LIN {X 0,Y 523.895,Z 313.853,A -85,B 0,C 180,E1 -4885.421,E2 -4885.421} C_VEL
LIN {X 0,Y 523.902,Z 313.843,A -85,B 0,C 180,E1 -4888.002,E2 -4888.002} C_VEL
LIN {X 0,Y 523.925,Z 313.85,A -85,B 0,C 180,E1 -4890.853,E2 -4890.853} C_VEL
LIN {X 0,Y 523.919,Z 313.846,A -85,B 0,C 180,E1 -4893.73,E2 -4893.73} C_VEL
LIN {X 0,Y 523.893,Z 313.85,A -85,B 0,C 180,E1 -4896.402,E2 -4896.402} C_VEL
LIN {X 0,Y 523.91,Z 313.85,A -85,B 0,C 180,E1 -4899.085,E2 -4899.085} C_VEL
LIN {X 0,Y 523.942,Z 313.841,A -85,B 0,C 180,E1 -4902.119,E2 -4902.119} C_VEL
LIN {X 0,Y 523.933,Z 313.845,A -85,B 0,C 180,E1 -4905.311,E2 -4905.311} C_VEL
LIN {X 0,Y 523.907,Z 313.852,A -85,B 0,C 180,E1 -4906.866,E2 -4906.866} C_VEL
LIN {X 0,Y 523.227,Z 313.935,A -85,B 0,C 180,E1 -4907.294,E2 -4907.294} C_VEL
LIN {X 0,Y 520.387,Z 314.288,A -85,B 0,C 180,E1 -4907.962,E2 -4907.962} C_VEL
LIN {X 0,Y 517.542,Z 314.646,A -85,B 0,C 180,E1 -4908.638,E2 -4908.638} C_VEL
LIN {X 0,Y 516.872,Z 314.727,A -85,B 0,C 180,E1 -4909.074,E2 -4909.074} C_VEL
LIN {X 0,Y 516.91,Z 314.812,A -85,B 0,C 180,E1 -4909.879,E2 -4909.879} C_VEL
LIN {X 0,Y 518.209,Z 321.592,A -85,B 0,C 180,E1 -4911.166,E2 -4911.166} C_VEL
LIN {X 0,Y 518.031,Z 330.95,A -85,B 0,C 180,E1 -4912.826,E2 -4912.826} C_VEL
LIN {X 0,Y 518.003,Z 334.606,A -85,B 0,C 180,E1 -4913.443,E2 -4913.443} C_VEL
LIN {X 0,Y 520.419,Z 345.939,A -85,B 0,C 180,E1 -4913.696,E2 -4913.696} C_VEL
LIN {X 0,Y 519.712,Z 470.939,A -85,B 0,C 180,E1 -4915.474,E2 -4915.474} C_VEL
LIN {X 0,Y 519.472,Z 485.199,A -85,B 0,C 180,E1 -4915.836,E2 -4915.836} C_VEL
LIN {X 0,Y 519.165,Z 498.963,A -85,B 0,C 180,E1 -4916.347,E2 -4916.347} C_VEL
LIN {X 0,Y 518.789,Z 511.827,A -85,B 0,C 180,E1 -4916.982,E2 -4916.982} C_VEL
LIN {X 0,Y 518.377,Z 523.912,A -85,B 0,C 180,E1 -4917.736,E2 -4917.736} C_VEL
LIN {X 0,Y 517.97,Z 535.685,A -85,B 0,C 180,E1 -4918.645,E2 -4918.645} C_VEL
LIN {X 0,Y 517.554,Z 547.16,A -85,B 0,C 180,E1 -4919.727,E2 -4919.727} C_VEL
LIN {X 0,Y 517.208,Z 557.645,A -85,B 0,C 180,E1 -4920.937,E2 -4920.937} C_VEL
LIN {X 0,Y 516.873,Z 567.085,A -85,B 0,C 180,E1 -4922.278,E2 -4922.278} C_VEL
LIN {X 0,Y 516.634,Z 574.914,A -85,B 0,C 180,E1 -4923.646,E2 -4923.646} C_VEL
LIN {X 0,Y 516.429,Z 581.367,A -85,B 0,C 180,E1 -4925.048,E2 -4925.048} C_VEL
LIN {X 0,Y 516.394,Z 586.053,A -85,B 0,C 180,E1 -4926.33,E2 -4926.33} C_VEL
LIN {X 0,Y 516.291,Z 590.061,A -85,B 0,C 180,E1 -4927.765,E2 -4927.765} C_VEL
LIN {X 0,Y 516.188,Z 592.955,A -85,B 0,C 180,E1 -4929.269,E2 -4929.269} C_VEL
LIN {X 0,Y 516.2,Z 594.008,A -85,B 0,C 180,E1 -4930.101,E2 -4930.101} C_VEL
LIN {X 0,Y 516.169,Z 594.998,A -85,B 0,C 180,E1 -4931.751,E2 -4931.751} C_VEL
LIN {X 0,Y 516.164,Z 594.545,A -85,B 0,C 180,E1 -4933.386,E2 -4933.386} C_VEL
LIN {X 0,Y 516.216,Z 592.673,A -85,B 0,C 180,E1 -4935.009,E2 -4935.009} C_VEL
LIN {X 0,Y 516.273,Z 589.339,A -85,B 0,C 180,E1 -4936.62,E2 -4936.62} C_VEL
LIN {X 0,Y 516.396,Z 584.476,A -85,B 0,C 180,E1 -4938.221,E2 -4938.221} C_VEL
LIN {X 0,Y 516.474,Z 579.801,A -85,B 0,C 180,E1 -4939.415,E2 -4939.415} C_VEL
LIN {X 0,Y 516.689,Z 572.998,A -85,B 0,C 180,E1 -4940.804,E2 -4940.804} C_VEL
LIN {X 0,Y 516.94,Z 564.592,A -85,B 0,C 180,E1 -4942.187,E2 -4942.187} C_VEL
LIN {X 0,Y 517.273,Z 555.841,A -85,B 0,C 180,E1 -4943.369,E2 -4943.369} C_VEL
LIN {X 0,Y 517.611,Z 545.305,A -85,B 0,C 180,E1 -4944.547,E2 -4944.547} C_VEL
LIN {X 0,Y 517.958,Z 534.696,A -85,B 0,C 180,E1 -4945.526,E2 -4945.526} C_VEL
LIN {X 0,Y 518.401,Z 523.103,A -85,B 0,C 180,E1 -4946.406,E2 -4946.406} C_VEL
LIN {X 0,Y 518.815,Z 510.389,A -85,B 0,C 180,E1 -4947.186,E2 -4947.186} C_VEL
LIN {X 0,Y 519.208,Z 497.174,A -85,B 0,C 180,E1 -4947.819,E2 -4947.819} C_VEL
LIN {X 0,Y 519.498,Z 483.55,A -85,B 0,C 180,E1 -4948.305,E2 -4948.305} C_VEL
LIN {X 0,Y 519.723,Z 469.332,A -85,B 0,C 180,E1 -4948.645,E2 -4948.645} C_VEL
LIN {X 0,Y 520.457,Z 346.248,A -85,B 0,C 180,E1 -4950.386,E2 -4950.386} C_VEL
LIN {X 0,Y 517.964,Z 334.247,A -85,B 0,C 180,E1 -4950.669,E2 -4950.669} C_VEL
LIN {X 0,Y 518.252,Z 321.48,A -85,B 0,C 180,E1 -4952.916,E2 -4952.916} C_VEL
LIN {X 0,Y 516.918,Z 314.722,A -85,B 0,C 180,E1 -4954.216,E2 -4954.216} C_VEL
LIN {X 0,Y 516.981,Z 314.712,A -85,B 0,C 180,E1 -4956.244,E2 -4956.244} C_VEL
LIN {X 0,Y 516.932,Z 314.723,A -85,B 0,C 180,E1 -4959.39,E2 -4959.39} C_VEL
LIN {X 0,Y 516.95,Z 314.714,A -85,B 0,C 180,E1 -4961.807,E2 -4961.807} C_VEL
LIN {X 0,Y 516.934,Z 314.721,A -85,B 0,C 180,E1 -4965.143,E2 -4965.143} C_VEL
LIN {X 0,Y 516.91,Z 314.716,A -85,B 0,C 180,E1 -4968.223,E2 -4968.223} C_VEL
LIN {X 0,Y 516.902,Z 314.72,A -85,B 0,C 180,E1 -4970.702,E2 -4970.702} C_VEL
LIN {X 0,Y 516.882,Z 314.72,A -85,B 0,C 180,E1 -4974.074,E2 -4974.074} C_VEL
LIN {X 0,Y 516.835,Z 314.729,A -85,B 0,C 180,E1 -4976.663,E2 -4976.663} C_VEL
LIN {X 0,Y 516.878,Z 314.722,A -85,B 0,C 180,E1 -4979.518,E2 -4979.518} C_VEL
LIN {X 0,Y 516.862,Z 314.725,A -85,B 0,C 180,E1 -4982.538,E2 -4982.538} C_VEL
LIN {X 0,Y 516.847,Z 314.727,A -85,B 0,C 180,E1 -4985.327,E2 -4985.327} C_VEL
LIN {X 0,Y 516.859,Z 314.73,A -85,B 0,C 180,E1 -4988.718,E2 -4988.718} C_VEL
LIN {X 0,Y 516.841,Z 314.725,A -85,B 0,C 180,E1 -4991.783,E2 -4991.783} C_VEL
LIN {X 0,Y 516.895,Z 314.723,A -85,B 0,C 180,E1 -4995.007,E2 -4995.007} C_VEL
LIN {X 0,Y 516.845,Z 314.729,A -85,B 0,C 180,E1 -4998.408,E2 -4998.408} C_VEL
LIN {X 0,Y 516.854,Z 314.724,A -85,B 0,C 180,E1 -5001.282,E2 -5001.282} C_VEL
LIN {X 0,Y 516.849,Z 314.732,A -85,B 0,C 180,E1 -5004.674,E2 -5004.674} C_VEL
LIN {X 0,Y 516.892,Z 314.719,A -85,B 0,C 180,E1 -5007.458,E2 -5007.458} C_VEL
LIN {X 0,Y 516.889,Z 314.725,A -85,B 0,C 180,E1 -5010.694,E2 -5010.694} C_VEL
LIN {X 0,Y 516.879,Z 314.721,A -85,B 0,C 180,E1 -5013.819,E2 -5013.819} C_VEL
LIN {X 0,Y 516.842,Z 314.728,A -85,B 0,C 180,E1 -5016.775,E2 -5016.775} C_VEL
LIN {X 0,Y 516.928,Z 314.716,A -85,B 0,C 180,E1 -5019.736,E2 -5019.736} C_VEL
LIN {X 0,Y 516.866,Z 314.726,A -85,B 0,C 180,E1 -5022.594,E2 -5022.594} C_VEL
LIN {X 0,Y 516.934,Z 314.714,A -85,B 0,C 180,E1 -5025.03,E2 -5025.03} C_VEL
LIN {X 0,Y 516.969,Z 314.718,A -85,B 0,C 180,E1 -5028.234,E2 -5028.234} C_VEL
LIN {X 0,Y 516.955,Z 314.711,A -85,B 0,C 180,E1 -5031.4,E2 -5031.4} C_VEL
LIN {X 0,Y 517.02,Z 314.705,A -85,B 0,C 180,E1 -5034.54,E2 -5034.54} C_VEL
LIN {X 0,Y 517.082,Z 314.699,A -85,B 0,C 180,E1 -5037.663,E2 -5037.663} C_VEL
LIN {X 0,Y 517.093,Z 314.694,A -85,B 0,C 180,E1 -5040.779,E2 -5040.779} C_VEL
LIN {X 0,Y 516.976,Z 314.708,A -85,B 0,C 180,E1 -5043.117,E2 -5043.117} C_VEL
LIN {X 0,Y 516.991,Z 314.71,A -85,B 0,C 180,E1 -5046.244,E2 -5046.244} C_VEL
LIN {X 0,Y 516.967,Z 314.71,A -85,B 0,C 180,E1 -5048.601,E2 -5048.601} C_VEL
LIN {X 0,Y 516.955,Z 314.72,A -85,B 0,C 180,E1 -5051.807,E2 -5051.807} C_VEL
LIN {X 0,Y 516.948,Z 314.713,A -85,B 0,C 180,E1 -5055.146,E2 -5055.146} C_VEL
LIN {X 0,Y 516.928,Z 314.716,A -85,B 0,C 180,E1 -5058.222,E2 -5058.222} C_VEL
LIN {X 0,Y 516.916,Z 314.715,A -85,B 0,C 180,E1 -5060.702,E2 -5060.702} C_VEL
LIN {X 0,Y 516.894,Z 314.721,A -85,B 0,C 180,E1 -5064.073,E2 -5064.073} C_VEL
LIN {X 0,Y 516.926,Z 314.714,A -85,B 0,C 180,E1 -5066.658,E2 -5066.658} C_VEL
LIN {X 0,Y 516.914,Z 314.725,A -85,B 0,C 180,E1 -5069.524,E2 -5069.524} C_VEL
LIN {X 0,Y 516.899,Z 314.718,A -85,B 0,C 180,E1 -5072.543,E2 -5072.543} C_VEL
LIN {X 0,Y 516.868,Z 314.73,A -85,B 0,C 180,E1 -5075.329,E2 -5075.329} C_VEL
LIN {X 0,Y 516.882,Z 314.721,A -85,B 0,C 180,E1 -5077.943,E2 -5077.943} C_VEL
LIN {X 0,Y 516.887,Z 314.721,A -85,B 0,C 180,E1 -5080.742,E2 -5080.742} C_VEL
LIN {X 0,Y 516.887,Z 314.722,A -85,B 0,C 180,E1 -5082.831,E2 -5082.831} C_VEL
LIN {X 0,Y 516.927,Z 314.72,A -85,B 0,C 180,E1 -5085.01,E2 -5085.01} C_VEL
LIN {X 0,Y 516.917,Z 314.716,A -85,B 0,C 180,E1 -5088.399,E2 -5088.399} C_VEL
LIN {X 0,Y 516.886,Z 314.726,A -85,B 0,C 180,E1 -5091.284,E2 -5091.284} C_VEL
LIN {X 0,Y 516.876,Z 314.721,A -85,B 0,C 180,E1 -5094.219,E2 -5094.219} C_VEL
LIN {X 0,Y 516.899,Z 314.727,A -85,B 0,C 180,E1 -5097.053,E2 -5097.053} C_VEL
LIN {X 0,Y 516.891,Z 314.724,A -85,B 0,C 180,E1 -5099.796,E2 -5099.796} C_VEL
LIN {X 0,Y 516.926,Z 314.725,A -85,B 0,C 180,E1 -5102.905,E2 -5102.905} C_VEL
LIN {X 0,Y 516.96,Z 314.746,A -85,B 0,C 180,E1 -5103.344,E2 -5103.344} C_VEL
LIN {X 0,Y 519.314,Z 326.551,A -85,B 0,C 180,E1 -5105.195,E2 -5105.195} C_VEL
LIN {X 0,Y 518.6,Z 348.488,A -85,B 0,C 180,E1 -5108.328,E2 -5108.328} C_VEL
LIN {X 0,Y 518.011,Z 369.079,A -85,B 0,C 180,E1 -5111.222,E2 -5111.222} C_VEL
LIN {X 0,Y 518.022,Z 370.448,A -85,B 0,C 180,E1 -5111.379,E2 -5111.379} C_VEL
LIN {X 0,Y 520.349,Z 384.488,A -85,B 0,C 180,E1 -5111.665,E2 -5111.665} C_VEL
LIN {X 0,Y 519.632,Z 508.513,A -85,B 0,C 180,E1 -5113.423,E2 -5113.423} C_VEL
LIN {X 0,Y 519.349,Z 523,A -85,B 0,C 180,E1 -5113.788,E2 -5113.788} C_VEL
LIN {X 0,Y 519.043,Z 536.545,A -85,B 0,C 180,E1 -5114.287,E2 -5114.287} C_VEL
LIN {X 0,Y 518.616,Z 550.559,A -85,B 0,C 180,E1 -5114.979,E2 -5114.979} C_VEL
LIN {X 0,Y 518.19,Z 563.097,A -85,B 0,C 180,E1 -5115.769,E2 -5115.769} C_VEL
LIN {X 0,Y 517.789,Z 574.555,A -85,B 0,C 180,E1 -5116.659,E2 -5116.659} C_VEL
LIN {X 0,Y 517.429,Z 585.048,A -85,B 0,C 180,E1 -5117.643,E2 -5117.643} C_VEL
LIN {X 0,Y 517.129,Z 595.568,A -85,B 0,C 180,E1 -5118.833,E2 -5118.833} C_VEL
LIN {X 0,Y 516.807,Z 604.214,A -85,B 0,C 180,E1 -5120.015,E2 -5120.015} C_VEL
LIN {X 0,Y 516.591,Z 612.5,A -85,B 0,C 180,E1 -5121.393,E2 -5121.393} C_VEL
LIN {X 0,Y 516.447,Z 618.297,A -85,B 0,C 180,E1 -5122.571,E2 -5122.571} C_VEL
LIN {X 0,Y 516.365,Z 623.051,A -85,B 0,C 180,E1 -5123.748,E2 -5123.748} C_VEL
LIN {X 0,Y 516.306,Z 626.901,A -85,B 0,C 180,E1 -5124.923,E2 -5124.923} C_VEL
LIN {X 0,Y 516.325,Z 629.869,A -85,B 0,C 180,E1 -5126.097,E2 -5126.097} C_VEL
LIN {X 0,Y 516.259,Z 632.583,A -85,B 0,C 180,E1 -5127.659,E2 -5127.659} C_VEL
LIN {X 0,Y 516.157,Z 633.926,A -85,B 0,C 180,E1 -5129.219,E2 -5129.219} C_VEL
LIN {X 0,Y 516.157,Z 633.926,A -85,B 0,C 180,E1 -5130.779,E2 -5130.779} C_VEL
LIN {X 0,Y 516.259,Z 632.584,A -85,B 0,C 180,E1 -5132.34,E2 -5132.34} C_VEL
LIN {X 0,Y 516.324,Z 629.869,A -85,B 0,C 180,E1 -5133.902,E2 -5133.902} C_VEL
LIN {X 0,Y 516.366,Z 625.705,A -85,B 0,C 180,E1 -5135.466,E2 -5135.466} C_VEL
LIN {X 0,Y 516.401,Z 619.967,A -85,B 0,C 180,E1 -5137.035,E2 -5137.035} C_VEL
LIN {X 0,Y 516.582,Z 613.504,A -85,B 0,C 180,E1 -5138.409,E2 -5138.409} C_VEL
LIN {X 0,Y 516.76,Z 605.473,A -85,B 0,C 180,E1 -5139.787,E2 -5139.787} C_VEL
LIN {X 0,Y 517.069,Z 597.078,A -85,B 0,C 180,E1 -5140.969,E2 -5140.969} C_VEL
LIN {X 0,Y 517.388,Z 586.704,A -85,B 0,C 180,E1 -5142.183,E2 -5142.183} C_VEL
LIN {X 0,Y 517.738,Z 575.7,A -85,B 0,C 180,E1 -5143.241,E2 -5143.241} C_VEL
LIN {X 0,Y 518.14,Z 564.494,A -85,B 0,C 180,E1 -5144.131,E2 -5144.131} C_VEL
LIN {X 0,Y 518.543,Z 552.292,A -85,B 0,C 180,E1 -5144.922,E2 -5144.922} C_VEL
LIN {X 0,Y 518.966,Z 538.756,A -85,B 0,C 180,E1 -5145.613,E2 -5145.613} C_VEL
LIN {X 0,Y 519.283,Z 524.557,A -85,B 0,C 180,E1 -5146.159,E2 -5146.159} C_VEL
LIN {X 0,Y 519.563,Z 510.759,A -85,B 0,C 180,E1 -5146.527,E2 -5146.527} C_VEL
LIN {X 0,Y 519.766,Z 488.556,A -85,B 0,C 180,E1 -5146.874,E2 -5146.874} C_VEL
LIN {X 0,Y 520.331,Z 383.603,A -85,B 0,C 180,E1 -5148.347,E2 -5148.347} C_VEL
LIN {X 0,Y 517.954,Z 369.999,A -85,B 0,C 180,E1 -5148.634,E2 -5148.634} C_VEL
LIN {X 0,Y 518.61,Z 348.337,A -85,B 0,C 180,E1 -5151.67,E2 -5151.67} C_VEL
LIN {X 0,Y 519.25,Z 327.875,A -85,B 0,C 180,E1 -5154.594,E2 -5154.594} C_VEL
LIN {X 0,Y 518.84,Z 323.477,A -85,B 0,C 180,E1 -5155.256,E2 -5155.256} C_VEL
LIN {X 0,Y 516.957,Z 314.718,A -85,B 0,C 180,E1 -5156.655,E2 -5156.655} C_VEL
LIN {X 0,Y 516.909,Z 314.722,A -85,B 0,C 180,E1 -5159.523,E2 -5159.523} C_VEL
LIN {X 0,Y 516.895,Z 314.723,A -85,B 0,C 180,E1 -5162.543,E2 -5162.543} C_VEL
LIN {X 0,Y 516.88,Z 314.723,A -85,B 0,C 180,E1 -5165.331,E2 -5165.331} C_VEL
LIN {X 0,Y 516.878,Z 314.722,A -85,B 0,C 180,E1 -5167.942,E2 -5167.942} C_VEL
LIN {X 0,Y 516.9,Z 314.726,A -85,B 0,C 180,E1 -5170.739,E2 -5170.739} C_VEL
LIN {X 0,Y 516.878,Z 314.723,A -85,B 0,C 180,E1 -5173.902,E2 -5173.902} C_VEL
LIN {X 0,Y 516.878,Z 314.719,A -85,B 0,C 180,E1 -5176.106,E2 -5176.106} C_VEL
LIN {X 0,Y 516.912,Z 314.723,A -85,B 0,C 180,E1 -5178.397,E2 -5178.397} C_VEL
LIN {X 0,Y 516.877,Z 314.72,A -85,B 0,C 180,E1 -5181.284,E2 -5181.284} C_VEL
LIN {X 0,Y 516.883,Z 314.726,A -85,B 0,C 180,E1 -5184.22,E2 -5184.22} C_VEL
LIN {X 0,Y 516.89,Z 314.719,A -85,B 0,C 180,E1 -5187.052,E2 -5187.052} C_VEL
LIN {X 0,Y 516.895,Z 314.72,A -85,B 0,C 180,E1 -5189.796,E2 -5189.796} C_VEL
LIN {X 0,Y 516.924,Z 314.72,A -85,B 0,C 180,E1 -5192.467,E2 -5192.467} C_VEL
LIN {X 0,Y 516.897,Z 314.719,A -85,B 0,C 180,E1 -5195.071,E2 -5195.071} C_VEL
LIN {X 0,Y 516.878,Z 314.726,A -85,B 0,C 180,E1 -5198.462,E2 -5198.462} C_VEL
LIN {X 0,Y 516.894,Z 314.716,A -85,B 0,C 180,E1 -5200.954,E2 -5200.954} C_VEL
LIN {X 0,Y 516.904,Z 314.719,A -85,B 0,C 180,E1 -5203.41,E2 -5203.41} C_VEL
LIN {X 0,Y 516.885,Z 314.723,A -85,B 0,C 180,E1 -5205.833,E2 -5205.833} C_VEL
LIN {X 0,Y 516.957,Z 314.713,A -85,B 0,C 180,E1 -5208.233,E2 -5208.233} C_VEL
LIN {X 0,Y 516.954,Z 314.714,A -85,B 0,C 180,E1 -5211.399,E2 -5211.399} C_VEL
LIN {X 0,Y 516.989,Z 314.711,A -85,B 0,C 180,E1 -5213.756,E2 -5213.756} C_VEL
LIN {X 0,Y 516.962,Z 314.708,A -85,B 0,C 180,E1 -5216.883,E2 -5216.883} C_VEL
LIN {X 0,Y 517.08,Z 314.698,A -85,B 0,C 180,E1 -5219.221,E2 -5219.221} C_VEL
LIN {X 0,Y 517.063,Z 314.699,A -85,B 0,C 180,E1 -5222.337,E2 -5222.337} C_VEL
LIN {X 0,Y 516.97,Z 314.714,A -85,B 0,C 180,E1 -5225.46,E2 -5225.46} C_VEL
LIN {X 0,Y 516.914,Z 314.715,A -85,B 0,C 180,E1 -5228.601,E2 -5228.601} C_VEL
LIN {X 0,Y 516.942,Z 314.715,A -85,B 0,C 180,E1 -5231.807,E2 -5231.807} C_VEL
LIN {X 0,Y 516.924,Z 314.721,A -85,B 0,C 180,E1 -5235.142,E2 -5235.142} C_VEL
LIN {X 0,Y 516.865,Z 314.723,A -85,B 0,C 180,E1 -5238.224,E2 -5238.224} C_VEL
LIN {X 0,Y 516.89,Z 314.721,A -85,B 0,C 180,E1 -5240.702,E2 -5240.702} C_VEL
LIN {X 0,Y 516.845,Z 314.733,A -85,B 0,C 180,E1 -5243.224,E2 -5243.224} C_VEL
LIN {X 0,Y 516.888,Z 314.721,A -85,B 0,C 180,E1 -5246.186,E2 -5246.186} C_VEL
LIN {X 0,Y 516.893,Z 314.724,A -85,B 0,C 180,E1 -5249.306,E2 -5249.306} C_VEL
LIN {X 0,Y 516.884,Z 314.724,A -85,B 0,C 180,E1 -5252.543,E2 -5252.543} C_VEL
LIN {X 0,Y 516.855,Z 314.729,A -85,B 0,C 180,E1 -5255.33,E2 -5255.33} C_VEL
LIN {X 0,Y 516.87,Z 314.724,A -85,B 0,C 180,E1 -5257.943,E2 -5257.943} C_VEL
LIN {X 0,Y 516.874,Z 314.728,A -85,B 0,C 180,E1 -5260.742,E2 -5260.742} C_VEL
LIN {X 0,Y 516.873,Z 314.73,A -85,B 0,C 180,E1 -5262.832,E2 -5262.832} C_VEL
LIN {X 0,Y 516.886,Z 314.726,A -85,B 0,C 180,E1 -5265.007,E2 -5265.007} C_VEL
LIN {X 0,Y 516.905,Z 314.725,A -85,B 0,C 180,E1 -5268.399,E2 -5268.399} C_VEL
LIN {X 0,Y 516.872,Z 314.727,A -85,B 0,C 180,E1 -5269.074,E2 -5269.074} C_VEL
LIN {X 0,Y 516.621,Z 315.183,A -85,B 0,C 180,E1 -5269.504,E2 -5269.504} C_VEL
LIN {X 0,Y 515.985,Z 316.355,A -85,B 0,C 180,E1 -5269.915,E2 -5269.915} C_VEL
LIN {X 0,Y 514.111,Z 320.017,A -85,B 0,C 180,E1 -5270.678,E2 -5270.678} C_VEL
LIN {X 0,Y 511.532,Z 326.847,A -85,B 0,C 180,E1 -5271.783,E2 -5271.783} C_VEL
LIN {X 0,Y 511.257,Z 329.026,A -85,B 0,C 180,E1 -5272.164,E2 -5272.164} C_VEL
LIN {X 0,Y 511.074,Z 334.779,A -85,B 0,C 180,E1 -5273.179,E2 -5273.179} C_VEL
LIN {X 0,Y 513.686,Z 346.942,A -85,B 0,C 180,E1 -5273.458,E2 -5273.458} C_VEL
LIN {X 0,Y 512.919,Z 471.171,A -85,B 0,C 180,E1 -5275.249,E2 -5275.249} C_VEL
LIN {X 0,Y 512.66,Z 485.216,A -85,B 0,C 180,E1 -5275.608,E2 -5275.608} C_VEL
LIN {X 0,Y 512.349,Z 499.236,A -85,B 0,C 180,E1 -5276.135,E2 -5276.135} C_VEL
LIN {X 0,Y 511.895,Z 513.153,A -85,B 0,C 180,E1 -5276.836,E2 -5276.836} C_VEL
LIN {X 0,Y 511.478,Z 524.978,A -85,B 0,C 180,E1 -5277.597,E2 -5277.597} C_VEL
LIN {X 0,Y 511.033,Z 536.424,A -85,B 0,C 180,E1 -5278.501,E2 -5278.501} C_VEL
LIN {X 0,Y 510.588,Z 547.892,A -85,B 0,C 180,E1 -5279.606,E2 -5279.606} C_VEL
LIN {X 0,Y 510.249,Z 557.474,A -85,B 0,C 180,E1 -5280.729,E2 -5280.729} C_VEL
LIN {X 0,Y 509.903,Z 566.821,A -85,B 0,C 180,E1 -5282.056,E2 -5282.056} C_VEL
LIN {X 0,Y 509.617,Z 574.325,A -85,B 0,C 180,E1 -5283.358,E2 -5283.358} C_VEL
LIN {X 0,Y 509.427,Z 580.551,A -85,B 0,C 180,E1 -5284.681,E2 -5284.681} C_VEL
LIN {X 0,Y 509.321,Z 585.551,A -85,B 0,C 180,E1 -5286.006,E2 -5286.006} C_VEL
LIN {X 0,Y 509.189,Z 590.165,A -85,B 0,C 180,E1 -5287.63,E2 -5287.63} C_VEL
LIN {X 0,Y 509.119,Z 592.842,A -85,B 0,C 180,E1 -5288.968,E2 -5288.968} C_VEL
LIN {X 0,Y 509.121,Z 594.033,A -85,B 0,C 180,E1 -5289.831,E2 -5289.831} C_VEL
LIN {X 0,Y 509.085,Z 595.215,A -85,B 0,C 180,E1 -5291.488,E2 -5291.488} C_VEL
LIN {X 0,Y 509.128,Z 595.268,A -85,B 0,C 180,E1 -5292.322,E2 -5292.322} C_VEL
LIN {X 0,Y 509.046,Z 594.314,A -85,B 0,C 180,E1 -5293.972,E2 -5293.972} C_VEL
LIN {X 0,Y 509.161,Z 591.933,A -85,B 0,C 180,E1 -5295.615,E2 -5295.615} C_VEL
LIN {X 0,Y 509.238,Z 588.114,A -85,B 0,C 180,E1 -5297.244,E2 -5297.244} C_VEL
LIN {X 0,Y 509.344,Z 584.322,A -85,B 0,C 180,E1 -5298.424,E2 -5298.424} C_VEL
LIN {X 0,Y 509.455,Z 579.375,A -85,B 0,C 180,E1 -5299.67,E2 -5299.67} C_VEL
LIN {X 0,Y 509.635,Z 572.43,A -85,B 0,C 180,E1 -5301.076,E2 -5301.076} C_VEL
LIN {X 0,Y 509.973,Z 563.568,A -85,B 0,C 180,E1 -5302.518,E2 -5302.518} C_VEL
LIN {X 0,Y 510.304,Z 554.893,A -85,B 0,C 180,E1 -5303.675,E2 -5303.675} C_VEL
LIN {X 0,Y 510.717,Z 544.106,A -85,B 0,C 180,E1 -5304.869,E2 -5304.869} C_VEL
LIN {X 0,Y 511.111,Z 533.199,A -85,B 0,C 180,E1 -5305.861,E2 -5305.861} C_VEL
LIN {X 0,Y 511.596,Z 521.209,A -85,B 0,C 180,E1 -5306.752,E2 -5306.752} C_VEL
LIN {X 0,Y 512.078,Z 507.819,A -85,B 0,C 180,E1 -5307.543,E2 -5307.543} C_VEL
LIN {X 0,Y 512.445,Z 494.913,A -85,B 0,C 180,E1 -5308.134,E2 -5308.134} C_VEL
LIN {X 0,Y 512.725,Z 481.071,A -85,B 0,C 180,E1 -5308.602,E2 -5308.602} C_VEL
LIN {X 0,Y 512.975,Z 466.261,A -85,B 0,C 180,E1 -5308.925,E2 -5308.925} C_VEL
LIN {X 0,Y 513.668,Z 347.031,A -85,B 0,C 180,E1 -5310.63,E2 -5310.63} C_VEL
LIN {X 0,Y 511.048,Z 334.459,A -85,B 0,C 180,E1 -5310.936,E2 -5310.936} C_VEL
LIN {X 0,Y 511.341,Z 323.112,A -85,B 0,C 180,E1 -5312.955,E2 -5312.955} C_VEL
LIN {X 0,Y 509.902,Z 315.596,A -85,B 0,C 180,E1 -5314.398,E2 -5314.398} C_VEL
LIN {X 0,Y 509.973,Z 315.587,A -85,B 0,C 180,E1 -5317.145,E2 -5317.145} C_VEL
LIN {X 0,Y 509.843,Z 315.6,A -85,B 0,C 180,E1 -5320.324,E2 -5320.324} C_VEL
LIN {X 0,Y 509.867,Z 315.596,A -85,B 0,C 180,E1 -5322.742,E2 -5322.742} C_VEL
LIN {X 0,Y 509.843,Z 315.597,A -85,B 0,C 180,E1 -5326.004,E2 -5326.004} C_VEL
LIN {X 0,Y 509.855,Z 315.596,A -85,B 0,C 180,E1 -5328.485,E2 -5328.485} C_VEL
LIN {X 0,Y 509.843,Z 315.603,A -85,B 0,C 180,E1 -5331.003,E2 -5331.003} C_VEL
LIN {X 0,Y 509.816,Z 315.603,A -85,B 0,C 180,E1 -5333.565,E2 -5333.565} C_VEL
LIN {X 0,Y 509.812,Z 315.601,A -85,B 0,C 180,E1 -5336.357,E2 -5336.357} C_VEL
LIN {X 0,Y 509.829,Z 315.605,A -85,B 0,C 180,E1 -5338.848,E2 -5338.848} C_VEL
LIN {X 0,Y 509.786,Z 315.605,A -85,B 0,C 180,E1 -5341.593,E2 -5341.593} C_VEL
LIN {X 0,Y 509.826,Z 315.601,A -85,B 0,C 180,E1 -5344.416,E2 -5344.416} C_VEL
LIN {X 0,Y 509.773,Z 315.608,A -85,B 0,C 180,E1 -5347.345,E2 -5347.345} C_VEL
LIN {X 0,Y 509.811,Z 315.604,A -85,B 0,C 180,E1 -5350.385,E2 -5350.385} C_VEL
LIN {X 0,Y 509.789,Z 315.604,A -85,B 0,C 180,E1 -5353.576,E2 -5353.576} C_VEL
LIN {X 0,Y 509.789,Z 315.608,A -85,B 0,C 180,E1 -5356.425,E2 -5356.425} C_VEL
LIN {X 0,Y 509.791,Z 315.603,A -85,B 0,C 180,E1 -5359.614,E2 -5359.614} C_VEL
LIN {X 0,Y 509.772,Z 315.614,A -85,B 0,C 180,E1 -5362.656,E2 -5362.656} C_VEL
LIN {X 0,Y 509.838,Z 315.598,A -85,B 0,C 180,E1 -5365.801,E2 -5365.801} C_VEL
LIN {X 0,Y 509.837,Z 315.603,A -85,B 0,C 180,E1 -5368.722,E2 -5368.722} C_VEL
LIN {X 0,Y 509.823,Z 315.6,A -85,B 0,C 180,E1 -5371.153,E2 -5371.153} C_VEL
LIN {X 0,Y 509.848,Z 315.597,A -85,B 0,C 180,E1 -5373.826,E2 -5373.826} C_VEL
LIN {X 0,Y 509.809,Z 315.609,A -85,B 0,C 180,E1 -5376.436,E2 -5376.436} C_VEL
LIN {X 0,Y 509.906,Z 315.591,A -85,B 0,C 180,E1 -5379.845,E2 -5379.845} C_VEL
LIN {X 0,Y 509.848,Z 315.604,A -85,B 0,C 180,E1 -5382.347,E2 -5382.347} C_VEL
LIN {X 0,Y 509.885,Z 315.593,A -85,B 0,C 180,E1 -5384.818,E2 -5384.818} C_VEL
LIN {X 0,Y 509.903,Z 315.597,A -85,B 0,C 180,E1 -5388.125,E2 -5388.125} C_VEL
LIN {X 0,Y 509.903,Z 315.589,A -85,B 0,C 180,E1 -5391.28,E2 -5391.28} C_VEL
LIN {X 0,Y 509.971,Z 315.584,A -85,B 0,C 180,E1 -5394.464,E2 -5394.464} C_VEL
LIN {X 0,Y 510.052,Z 315.574,A -85,B 0,C 180,E1 -5397.631,E2 -5397.631} C_VEL
LIN {X 0,Y 510.063,Z 315.57,A -85,B 0,C 180,E1 -5400.79,E2 -5400.79} C_VEL
LIN {X 0,Y 509.92,Z 315.587,A -85,B 0,C 180,E1 -5403.161,E2 -5403.161} C_VEL
LIN {X 0,Y 509.939,Z 315.588,A -85,B 0,C 180,E1 -5406.33,E2 -5406.33} C_VEL
LIN {X 0,Y 509.913,Z 315.588,A -85,B 0,C 180,E1 -5408.72,E2 -5408.72} C_VEL
LIN {X 0,Y 509.908,Z 315.595,A -85,B 0,C 180,E1 -5411.932,E2 -5411.932} C_VEL
LIN {X 0,Y 509.898,Z 315.592,A -85,B 0,C 180,E1 -5415.242,E2 -5415.242} C_VEL
LIN {X 0,Y 509.885,Z 315.596,A -85,B 0,C 180,E1 -5417.998,E2 -5417.998} C_VEL
LIN {X 0,Y 509.854,Z 315.596,A -85,B 0,C 180,E1 -5421.002,E2 -5421.002} C_VEL
LIN {X 0,Y 509.826,Z 315.607,A -85,B 0,C 180,E1 -5423.564,E2 -5423.564} C_VEL
LIN {X 0,Y 509.914,Z 315.588,A -85,B 0,C 180,E1 -5426.378,E2 -5426.378} C_VEL
LIN {X 0,Y 509.878,Z 315.593,A -85,B 0,C 180,E1 -5428.844,E2 -5428.844} C_VEL
LIN {X 0,Y 509.824,Z 315.606,A -85,B 0,C 180,E1 -5431.59,E2 -5431.59} C_VEL
LIN {X 0,Y 509.85,Z 315.596,A -85,B 0,C 180,E1 -5434.414,E2 -5434.414} C_VEL
LIN {X 0,Y 509.811,Z 315.609,A -85,B 0,C 180,E1 -5437.342,E2 -5437.342} C_VEL
LIN {X 0,Y 509.842,Z 315.597,A -85,B 0,C 180,E1 -5440.382,E2 -5440.382} C_VEL
LIN {X 0,Y 509.828,Z 315.604,A -85,B 0,C 180,E1 -5443.062,E2 -5443.062} C_VEL
LIN {X 0,Y 509.834,Z 315.599,A -85,B 0,C 180,E1 -5445.792,E2 -5445.792} C_VEL
LIN {X 0,Y 509.859,Z 315.596,A -85,B 0,C 180,E1 -5448.574,E2 -5448.574} C_VEL
LIN {X 0,Y 509.855,Z 315.596,A -85,B 0,C 180,E1 -5451.786,E2 -5451.786} C_VEL
LIN {X 0,Y 509.835,Z 315.6,A -85,B 0,C 180,E1 -5454.622,E2 -5454.622} C_VEL
LIN {X 0,Y 509.865,Z 315.6,A -85,B 0,C 180,E1 -5457.481,E2 -5457.481} C_VEL
LIN {X 0,Y 509.862,Z 315.6,A -85,B 0,C 180,E1 -5460.274,E2 -5460.274} C_VEL
LIN {X 0,Y 509.911,Z 315.608,A -85,B 0,C 180,E1 -5463.116,E2 -5463.116} C_VEL
LIN {X 0,Y 512.392,Z 327.624,A -85,B 0,C 180,E1 -5465.034,E2 -5465.034} C_VEL
LIN {X 0,Y 511.764,Z 346.778,A -85,B 0,C 180,E1 -5467.811,E2 -5467.811} C_VEL
LIN {X 0,Y 511.165,Z 367.213,A -85,B 0,C 180,E1 -5470.732,E2 -5470.732} C_VEL
LIN {X 0,Y 511.049,Z 370.036,A -85,B 0,C 180,E1 -5471.114,E2 -5471.114} C_VEL
LIN {X 0,Y 513.603,Z 385.193,A -85,B 0,C 180,E1 -5471.429,E2 -5471.429} C_VEL
LIN {X 0,Y 512.803,Z 508.183,A -85,B 0,C 180,E1 -5473.196,E2 -5473.196} C_VEL
LIN {X 0,Y 512.514,Z 522.519,A -85,B 0,C 180,E1 -5473.56,E2 -5473.56} C_VEL
LIN {X 0,Y 512.181,Z 536.248,A -85,B 0,C 180,E1 -5474.071,E2 -5474.071} C_VEL
LIN {X 0,Y 511.732,Z 550.27,A -85,B 0,C 180,E1 -5474.772,E2 -5474.772} C_VEL
LIN {X 0,Y 511.266,Z 562.812,A -85,B 0,C 180,E1 -5475.572,E2 -5475.572} C_VEL
LIN {X 0,Y 510.808,Z 574.273,A -85,B 0,C 180,E1 -5476.473,E2 -5476.473} C_VEL
LIN {X 0,Y 510.446,Z 584.995,A -85,B 0,C 180,E1 -5477.494,E2 -5477.494} C_VEL
LIN {X 0,Y 510.1,Z 595.291,A -85,B 0,C 180,E1 -5478.677,E2 -5478.677} C_VEL
LIN {X 0,Y 509.745,Z 603.94,A -85,B 0,C 180,E1 -5479.875,E2 -5479.875} C_VEL
LIN {X 0,Y 509.536,Z 612.229,A -85,B 0,C 180,E1 -5481.273,E2 -5481.273} C_VEL
LIN {X 0,Y 509.37,Z 618.026,A -85,B 0,C 180,E1 -5482.468,E2 -5482.468} C_VEL
LIN {X 0,Y 509.262,Z 622.781,A -85,B 0,C 180,E1 -5483.661,E2 -5483.661} C_VEL
LIN {X 0,Y 509.236,Z 626.634,A -85,B 0,C 180,E1 -5484.853,E2 -5484.853} C_VEL
LIN {X 0,Y 509.218,Z 629.601,A -85,B 0,C 180,E1 -5486.042,E2 -5486.042} C_VEL
LIN {X 0,Y 509.188,Z 632.317,A -85,B 0,C 180,E1 -5487.626,E2 -5487.626} C_VEL
LIN {X 0,Y 509.071,Z 633.658,A -85,B 0,C 180,E1 -5489.208,E2 -5489.208} C_VEL
LIN {X 0,Y 509.071,Z 633.657,A -85,B 0,C 180,E1 -5490.79,E2 -5490.79} C_VEL
LIN {X 0,Y 509.187,Z 632.314,A -85,B 0,C 180,E1 -5492.372,E2 -5492.372} C_VEL
LIN {X 0,Y 509.218,Z 629.596,A -85,B 0,C 180,E1 -5493.956,E2 -5493.956} C_VEL
LIN {X 0,Y 509.282,Z 625.43,A -85,B 0,C 180,E1 -5495.543,E2 -5495.543} C_VEL
LIN {X 0,Y 509.326,Z 619.689,A -85,B 0,C 180,E1 -5497.133,E2 -5497.133} C_VEL
LIN {X 0,Y 509.504,Z 613.222,A -85,B 0,C 180,E1 -5498.527,E2 -5498.527} C_VEL
LIN {X 0,Y 509.723,Z 605.188,A -85,B 0,C 180,E1 -5499.924,E2 -5499.924} C_VEL
LIN {X 0,Y 510.028,Z 596.789,A -85,B 0,C 180,E1 -5501.122,E2 -5501.122} C_VEL
LIN {X 0,Y 510.402,Z 586.037,A -85,B 0,C 180,E1 -5502.393,E2 -5502.393} C_VEL
LIN {X 0,Y 510.781,Z 575.403,A -85,B 0,C 180,E1 -5503.425,E2 -5503.425} C_VEL
LIN {X 0,Y 511.224,Z 564.192,A -85,B 0,C 180,E1 -5504.326,E2 -5504.326} C_VEL
LIN {X 0,Y 511.646,Z 551.983,A -85,B 0,C 180,E1 -5505.128,E2 -5505.128} C_VEL
LIN {X 0,Y 512.119,Z 538.44,A -85,B 0,C 180,E1 -5505.827,E2 -5505.827} C_VEL
LIN {X 0,Y 512.458,Z 524.378,A -85,B 0,C 180,E1 -5506.375,E2 -5506.375} C_VEL
LIN {X 0,Y 512.742,Z 510.405,A -85,B 0,C 180,E1 -5506.753,E2 -5506.753} C_VEL
LIN {X 0,Y 512.957,Z 488.163,A -85,B 0,C 180,E1 -5507.105,E2 -5507.105} C_VEL
LIN {X 0,Y 513.613,Z 385.046,A -85,B 0,C 180,E1 -5508.57,E2 -5508.57} C_VEL
LIN {X 0,Y 511.047,Z 369.712,A -85,B 0,C 180,E1 -5508.896,E2 -5508.896} C_VEL
LIN {X 0,Y 511.705,Z 348.088,A -85,B 0,C 180,E1 -5511.978,E2 -5511.978} C_VEL
LIN {X 0,Y 512.383,Z 329.208,A -85,B 0,C 180,E1 -5514.715,E2 -5514.715} C_VEL
LIN {X 0,Y 511.866,Z 324.723,A -85,B 0,C 180,E1 -5515.407,E2 -5515.407} C_VEL
LIN {X 0,Y 509.903,Z 315.598,A -85,B 0,C 180,E1 -5516.925,E2 -5516.925} C_VEL
LIN {X 0,Y 509.855,Z 315.599,A -85,B 0,C 180,E1 -5519.75,E2 -5519.75} C_VEL
LIN {X 0,Y 509.872,Z 315.601,A -85,B 0,C 180,E1 -5522.773,E2 -5522.773} C_VEL
LIN {X 0,Y 509.84,Z 315.598,A -85,B 0,C 180,E1 -5525.58,E2 -5525.58} C_VEL
LIN {X 0,Y 509.848,Z 315.6,A -85,B 0,C 180,E1 -5528.337,E2 -5528.337} C_VEL
LIN {X 0,Y 509.861,Z 315.594,A -85,B 0,C 180,E1 -5531.424,E2 -5531.424} C_VEL
LIN {X 0,Y 509.852,Z 315.602,A -85,B 0,C 180,E1 -5534.667,E2 -5534.667} C_VEL
LIN {X 0,Y 509.856,Z 315.599,A -85,B 0,C 180,E1 -5538.102,E2 -5538.102} C_VEL
LIN {X 0,Y 509.842,Z 315.598,A -85,B 0,C 180,E1 -5540.647,E2 -5540.647} C_VEL
LIN {X 0,Y 509.829,Z 315.599,A -85,B 0,C 180,E1 -5543.647,E2 -5543.647} C_VEL
LIN {X 0,Y 509.855,Z 315.601,A -85,B 0,C 180,E1 -5546.539,E2 -5546.539} C_VEL
LIN {X 0,Y 509.844,Z 315.597,A -85,B 0,C 180,E1 -5549.334,E2 -5549.334} C_VEL
LIN {X 0,Y 509.889,Z 315.596,A -85,B 0,C 180,E1 -5552.054,E2 -5552.054} C_VEL
LIN {X 0,Y 509.867,Z 315.597,A -85,B 0,C 180,E1 -5554.703,E2 -5554.703} C_VEL
LIN {X 0,Y 509.818,Z 315.598,A -85,B 0,C 180,E1 -5557.457,E2 -5557.457} C_VEL
LIN {X 0,Y 509.909,Z 315.594,A -85,B 0,C 180,E1 -5559.844,E2 -5559.844} C_VEL
LIN {X 0,Y 509.875,Z 315.594,A -85,B 0,C 180,E1 -5563.174,E2 -5563.174} C_VEL
LIN {X 0,Y 509.854,Z 315.596,A -85,B 0,C 180,E1 -5565.634,E2 -5565.634} C_VEL
LIN {X 0,Y 509.903,Z 315.586,A -85,B 0,C 180,E1 -5568.874,E2 -5568.874} C_VEL
LIN {X 0,Y 509.941,Z 315.588,A -85,B 0,C 180,E1 -5572.078,E2 -5572.078} C_VEL
LIN {X 0,Y 509.965,Z 315.584,A -85,B 0,C 180,E1 -5574.464,E2 -5574.464} C_VEL
LIN {X 0,Y 510.036,Z 315.577,A -85,B 0,C 180,E1 -5577.631,E2 -5577.631} C_VEL
LIN {X 0,Y 510.022,Z 315.578,A -85,B 0,C 180,E1 -5580,E2 -5580} C_VEL
LIN {X 0,Y 510.034,Z 315.574,A -85,B 0,C 180,E1 -5582.369,E2 -5582.369} C_VEL
LIN {X 0,Y 509.922,Z 315.592,A -85,B 0,C 180,E1 -5585.536,E2 -5585.536} C_VEL
LIN {X 0,Y 509.866,Z 315.597,A -85,B 0,C 180,E1 -5587.923,E2 -5587.923} C_VEL
LIN {X 0,Y 509.896,Z 315.595,A -85,B 0,C 180,E1 -5591.126,E2 -5591.126} C_VEL
LIN {X 0,Y 509.828,Z 315.6,A -85,B 0,C 180,E1 -5594.367,E2 -5594.367} C_VEL
LIN {X 0,Y 509.808,Z 315.602,A -85,B 0,C 180,E1 -5596.828,E2 -5596.828} C_VEL
LIN {X 0,Y 509.896,Z 315.591,A -85,B 0,C 180,E1 -5600.156,E2 -5600.156} C_VEL
LIN {X 0,Y 509.807,Z 315.606,A -85,B 0,C 180,E1 -5603.564,E2 -5603.564} C_VEL
LIN {X 0,Y 509.865,Z 315.596,A -85,B 0,C 180,E1 -5606.37,E2 -5606.37} C_VEL
LIN {X 0,Y 509.841,Z 315.6,A -85,B 0,C 180,E1 -5609.752,E2 -5609.752} C_VEL
LIN {X 0,Y 509.857,Z 315.6,A -85,B 0,C 180,E1 -5612.773,E2 -5612.773} C_VEL
LIN {X 0,Y 509.815,Z 315.603,A -85,B 0,C 180,E1 -5615.579,E2 -5615.579} C_VEL
LIN {X 0,Y 509.84,Z 315.601,A -85,B 0,C 180,E1 -5618.338,E2 -5618.338} C_VEL
LIN {X 0,Y 509.846,Z 315.598,A -85,B 0,C 180,E1 -5621.426,E2 -5621.426} C_VEL
LIN {X 0,Y 509.83,Z 315.605,A -85,B 0,C 180,E1 -5624.67,E2 -5624.67} C_VEL
LIN {X 0,Y 509.824,Z 315.604,A -85,B 0,C 180,E1 -5627.511,E2 -5627.511} C_VEL
LIN {X 0,Y 509.858,Z 315.631,A -85,B 0,C 180,E1 -5629.658,E2 -5629.658} C_VEL
LIN {X 0,Y 511.337,Z 323.804,A -85,B 0,C 180,E1 -5631.226,E2 -5631.226} C_VEL
LIN {X 0,Y 511.257,Z 329.026,A -85,B 0,C 180,E1 -5632.164,E2 -5632.164} C_VEL
LIN {X 0,Y 511.04,Z 331.519,A -85,B 0,C 180,E1 -5632.494,E2 -5632.494} C_VEL
LIN {X 0,Y 510.231,Z 336.347,A -85,B 0,C 180,E1 -5632.855,E2 -5632.855} C_VEL
LIN {X 0,Y 509.152,Z 341.833,A -85,B 0,C 180,E1 -5633.081,E2 -5633.081} C_VEL
LIN {X 0,Y 507.698,Z 349.959,A -85,B 0,C 180,E1 -5633.252,E2 -5633.252} C_VEL
LIN {X 0,Y 506.97,Z 358.262,A -85,B 0,C 180,E1 -5633.364,E2 -5633.364} C_VEL
LIN {X 0,Y 506.13,Z 471.847,A -85,B 0,C 180,E1 -5635.028,E2 -5635.028} C_VEL
LIN {X 0,Y 505.856,Z 485.964,A -85,B 0,C 180,E1 -5635.398,E2 -5635.398} C_VEL
LIN {X 0,Y 505.53,Z 499.503,A -85,B 0,C 180,E1 -5635.915,E2 -5635.915} C_VEL
LIN {X 0,Y 505.074,Z 513.013,A -85,B 0,C 180,E1 -5636.603,E2 -5636.603} C_VEL
LIN {X 0,Y 504.62,Z 524.439,A -85,B 0,C 180,E1 -5637.339,E2 -5637.339} C_VEL
LIN {X 0,Y 504.114,Z 536.057,A -85,B 0,C 180,E1 -5638.257,E2 -5638.257} C_VEL
LIN {X 0,Y 503.706,Z 546.606,A -85,B 0,C 180,E1 -5639.27,E2 -5639.27} C_VEL
LIN {X 0,Y 503.287,Z 557.289,A -85,B 0,C 180,E1 -5640.513,E2 -5640.513} C_VEL
LIN {X 0,Y 502.926,Z 565.616,A -85,B 0,C 180,E1 -5641.687,E2 -5641.687} C_VEL
LIN {X 0,Y 502.623,Z 573.2,A -85,B 0,C 180,E1 -5642.972,E2 -5642.972} C_VEL
LIN {X 0,Y 502.402,Z 579.624,A -85,B 0,C 180,E1 -5644.301,E2 -5644.301} C_VEL
LIN {X 0,Y 502.278,Z 585.225,A -85,B 0,C 180,E1 -5645.75,E2 -5645.75} C_VEL
LIN {X 0,Y 502.171,Z 588.817,A -85,B 0,C 180,E1 -5646.93,E2 -5646.93} C_VEL
LIN {X 0,Y 502.098,Z 590.934,A -85,B 0,C 180,E1 -5647.796,E2 -5647.796} C_VEL
LIN {X 0,Y 502.031,Z 593.941,A -85,B 0,C 180,E1 -5649.515,E2 -5649.515} C_VEL
LIN {X 0,Y 501.999,Z 595.411,A -85,B 0,C 180,E1 -5651.217,E2 -5651.217} C_VEL
LIN {X 0,Y 502.046,Z 595.569,A -85,B 0,C 180,E1 -5652.158,E2 -5652.158} C_VEL
LIN {X 0,Y 501.976,Z 594.836,A -85,B 0,C 180,E1 -5653.74,E2 -5653.74} C_VEL
LIN {X 0,Y 502.074,Z 592.66,A -85,B 0,C 180,E1 -5655.407,E2 -5655.407} C_VEL
LIN {X 0,Y 502.165,Z 589.048,A -85,B 0,C 180,E1 -5657.061,E2 -5657.061} C_VEL
LIN {X 0,Y 502.311,Z 583.915,A -85,B 0,C 180,E1 -5658.705,E2 -5658.705} C_VEL
LIN {X 0,Y 502.437,Z 578.95,A -85,B 0,C 180,E1 -5659.931,E2 -5659.931} C_VEL
LIN {X 0,Y 502.651,Z 571.846,A -85,B 0,C 180,E1 -5661.356,E2 -5661.356} C_VEL
LIN {X 0,Y 502.996,Z 563.204,A -85,B 0,C 180,E1 -5662.758,E2 -5662.758} C_VEL
LIN {X 0,Y 503.387,Z 553.932,A -85,B 0,C 180,E1 -5663.99,E2 -5663.99} C_VEL
LIN {X 0,Y 503.806,Z 543.865,A -85,B 0,C 180,E1 -5665.099,E2 -5665.099} C_VEL
LIN {X 0,Y 504.248,Z 532.833,A -85,B 0,C 180,E1 -5666.105,E2 -5666.105} C_VEL
LIN {X 0,Y 504.747,Z 520.668,A -85,B 0,C 180,E1 -5667.008,E2 -5667.008} C_VEL
LIN {X 0,Y 505.258,Z 507.065,A -85,B 0,C 180,E1 -5667.809,E2 -5667.809} C_VEL
LIN {X 0,Y 505.658,Z 493.837,A -85,B 0,C 180,E1 -5668.408,E2 -5668.408} C_VEL
LIN {X 0,Y 505.976,Z 479.863,A -85,B 0,C 180,E1 -5668.869,E2 -5668.869} C_VEL
LIN {X 0,Y 506.2,Z 466.269,A -85,B 0,C 180,E1 -5669.161,E2 -5669.161} C_VEL
LIN {X 0,Y 506.995,Z 348.203,A -85,B 0,C 180,E1 -5670.87,E2 -5670.87} C_VEL
LIN {X 0,Y 504.131,Z 334.712,A -85,B 0,C 180,E1 -5671.199,E2 -5671.199} C_VEL
LIN {X 0,Y 504.455,Z 324.756,A -85,B 0,C 180,E1 -5672.995,E2 -5672.995} C_VEL
LIN {X 0,Y 502.831,Z 316.477,A -85,B 0,C 180,E1 -5674.61,E2 -5674.61} C_VEL
LIN {X 0,Y 502.931,Z 316.464,A -85,B 0,C 180,E1 -5677.226,E2 -5677.226} C_VEL
LIN {X 0,Y 502.802,Z 316.477,A -85,B 0,C 180,E1 -5680.47,E2 -5680.47} C_VEL
LIN {X 0,Y 502.818,Z 316.475,A -85,B 0,C 180,E1 -5682.923,E2 -5682.923} C_VEL
LIN {X 0,Y 502.847,Z 316.475,A -85,B 0,C 180,E1 -5685.4,E2 -5685.4} C_VEL
LIN {X 0,Y 502.82,Z 316.474,A -85,B 0,C 180,E1 -5688.753,E2 -5688.753} C_VEL
LIN {X 0,Y 502.779,Z 316.483,A -85,B 0,C 180,E1 -5691.312,E2 -5691.312} C_VEL
LIN {X 0,Y 502.763,Z 316.479,A -85,B 0,C 180,E1 -5693.916,E2 -5693.916} C_VEL
LIN {X 0,Y 502.781,Z 316.479,A -85,B 0,C 180,E1 -5696.571,E2 -5696.571} C_VEL
LIN {X 0,Y 502.788,Z 316.475,A -85,B 0,C 180,E1 -5699.93,E2 -5699.93} C_VEL
LIN {X 0,Y 502.768,Z 316.486,A -85,B 0,C 180,E1 -5703.037,E2 -5703.037} C_VEL
LIN {X 0,Y 502.743,Z 316.481,A -85,B 0,C 180,E1 -5705.954,E2 -5705.954} C_VEL
LIN {X 0,Y 502.775,Z 316.484,A -85,B 0,C 180,E1 -5708.979,E2 -5708.979} C_VEL
LIN {X 0,Y 502.744,Z 316.482,A -85,B 0,C 180,E1 -5712.192,E2 -5712.192} C_VEL
LIN {X 0,Y 502.776,Z 316.478,A -85,B 0,C 180,E1 -5715.472,E2 -5715.472} C_VEL
LIN {X 0,Y 502.756,Z 316.485,A -85,B 0,C 180,E1 -5718.928,E2 -5718.928} C_VEL
LIN {X 0,Y 502.751,Z 316.482,A -85,B 0,C 180,E1 -5722.043,E2 -5722.043} C_VEL
LIN {X 0,Y 502.782,Z 316.479,A -85,B 0,C 180,E1 -5725.033,E2 -5725.033} C_VEL
LIN {X 0,Y 502.778,Z 316.478,A -85,B 0,C 180,E1 -5727.915,E2 -5727.915} C_VEL
LIN {X 0,Y 502.785,Z 316.481,A -85,B 0,C 180,E1 -5730.71,E2 -5730.71} C_VEL
LIN {X 0,Y 502.774,Z 316.477,A -85,B 0,C 180,E1 -5733.46,E2 -5733.46} C_VEL
LIN {X 0,Y 502.761,Z 316.483,A -85,B 0,C 180,E1 -5736.085,E2 -5736.085} C_VEL
LIN {X 0,Y 502.831,Z 316.47,A -85,B 0,C 180,E1 -5739.464,E2 -5739.464} C_VEL
LIN {X 0,Y 502.8,Z 316.48,A -85,B 0,C 180,E1 -5742.091,E2 -5742.091} C_VEL
LIN {X 0,Y 502.828,Z 316.471,A -85,B 0,C 180,E1 -5745.429,E2 -5745.429} C_VEL
LIN {X 0,Y 502.878,Z 316.466,A -85,B 0,C 180,E1 -5748.717,E2 -5748.717} C_VEL
LIN {X 0,Y 502.874,Z 316.471,A -85,B 0,C 180,E1 -5751.967,E2 -5751.967} C_VEL
LIN {X 0,Y 502.925,Z 316.463,A -85,B 0,C 180,E1 -5754.387,E2 -5754.387} C_VEL
LIN {X 0,Y 503.02,Z 316.449,A -85,B 0,C 180,E1 -5757.598,E2 -5757.598} C_VEL
LIN {X 0,Y 503.013,Z 316.448,A -85,B 0,C 180,E1 -5760.801,E2 -5760.801} C_VEL
LIN {X 0,Y 503.02,Z 316.449,A -85,B 0,C 180,E1 -5762.403,E2 -5762.403} C_VEL
LIN {X 0,Y 502.928,Z 316.463,A -85,B 0,C 180,E1 -5765.614,E2 -5765.614} C_VEL
LIN {X 0,Y 502.872,Z 316.465,A -85,B 0,C 180,E1 -5768.844,E2 -5768.844} C_VEL
LIN {X 0,Y 502.849,Z 316.472,A -85,B 0,C 180,E1 -5772.102,E2 -5772.102} C_VEL
LIN {X 0,Y 502.852,Z 316.472,A -85,B 0,C 180,E1 -5775.4,E2 -5775.4} C_VEL
LIN {X 0,Y 502.844,Z 316.471,A -85,B 0,C 180,E1 -5778.12,E2 -5778.12} C_VEL
LIN {X 0,Y 502.833,Z 316.47,A -85,B 0,C 180,E1 -5780.536,E2 -5780.536} C_VEL
LIN {X 0,Y 502.791,Z 316.477,A -85,B 0,C 180,E1 -5783.041,E2 -5783.041} C_VEL
LIN {X 0,Y 502.825,Z 316.478,A -85,B 0,C 180,E1 -5785.677,E2 -5785.677} C_VEL
LIN {X 0,Y 502.842,Z 316.469,A -85,B 0,C 180,E1 -5788.373,E2 -5788.373} C_VEL
LIN {X 0,Y 502.797,Z 316.483,A -85,B 0,C 180,E1 -5791.499,E2 -5791.499} C_VEL
LIN {X 0,Y 502.807,Z 316.475,A -85,B 0,C 180,E1 -5793.994,E2 -5793.994} C_VEL
LIN {X 0,Y 502.768,Z 316.484,A -85,B 0,C 180,E1 -5797.176,E2 -5797.176} C_VEL
LIN {X 0,Y 502.791,Z 316.476,A -85,B 0,C 180,E1 -5800.015,E2 -5800.015} C_VEL
LIN {X 0,Y 502.807,Z 316.473,A -85,B 0,C 180,E1 -5802.199,E2 -5802.199} C_VEL
LIN {X 0,Y 502.805,Z 316.479,A -85,B 0,C 180,E1 -5805.468,E2 -5805.468} C_VEL
LIN {X 0,Y 502.823,Z 316.476,A -85,B 0,C 180,E1 -5808.934,E2 -5808.934} C_VEL
LIN {X 0,Y 502.797,Z 316.474,A -85,B 0,C 180,E1 -5812.046,E2 -5812.046} C_VEL
LIN {X 0,Y 502.804,Z 316.482,A -85,B 0,C 180,E1 -5815.034,E2 -5815.034} C_VEL
LIN {X 0,Y 502.786,Z 316.479,A -85,B 0,C 180,E1 -5817.915,E2 -5817.915} C_VEL
LIN {X 0,Y 502.827,Z 316.48,A -85,B 0,C 180,E1 -5820.712,E2 -5820.712} C_VEL
LIN {X 0,Y 502.876,Z 316.528,A -85,B 0,C 180,E1 -5822.898,E2 -5822.898} C_VEL
LIN {X 0,Y 505.264,Z 327.683,A -85,B 0,C 180,E1 -5824.706,E2 -5824.706} C_VEL
LIN {X 0,Y 505.443,Z 331.887,A -85,B 0,C 180,E1 -5825.345,E2 -5825.345} C_VEL
LIN {X 0,Y 504.718,Z 352.353,A -85,B 0,C 180,E1 -5828.345,E2 -5828.345} C_VEL
LIN {X 0,Y 504.132,Z 369.844,A -85,B 0,C 180,E1 -5830.846,E2 -5830.846} C_VEL
LIN {X 0,Y 506.884,Z 385.939,A -85,B 0,C 180,E1 -5831.189,E2 -5831.189} C_VEL
LIN {X 0,Y 506.018,Z 507.851,A -85,B 0,C 180,E1 -5832.964,E2 -5832.964} C_VEL
LIN {X 0,Y 505.683,Z 522.139,A -85,B 0,C 180,E1 -5833.329,E2 -5833.329} C_VEL
LIN {X 0,Y 505.342,Z 535.95,A -85,B 0,C 180,E1 -5833.85,E2 -5833.85} C_VEL
LIN {X 0,Y 504.853,Z 549.979,A -85,B 0,C 180,E1 -5834.559,E2 -5834.559} C_VEL
LIN {X 0,Y 504.341,Z 562.525,A -85,B 0,C 180,E1 -5835.37,E2 -5835.37} C_VEL
LIN {X 0,Y 503.802,Z 575.17,A -85,B 0,C 180,E1 -5836.384,E2 -5836.384} C_VEL
LIN {X 0,Y 503.407,Z 585.801,A -85,B 0,C 180,E1 -5837.43,E2 -5837.43} C_VEL
LIN {X 0,Y 503.002,Z 596.55,A -85,B 0,C 180,E1 -5838.719,E2 -5838.719} C_VEL
LIN {X 0,Y 502.677,Z 604.945,A -85,B 0,C 180,E1 -5839.934,E2 -5839.934} C_VEL
LIN {X 0,Y 502.427,Z 612.973,A -85,B 0,C 180,E1 -5841.351,E2 -5841.351} C_VEL
LIN {X 0,Y 502.252,Z 619.439,A -85,B 0,C 180,E1 -5842.764,E2 -5842.764} C_VEL
LIN {X 0,Y 502.198,Z 625.174,A -85,B 0,C 180,E1 -5844.378,E2 -5844.378} C_VEL
LIN {X 0,Y 502.114,Z 629.332,A -85,B 0,C 180,E1 -5845.986,E2 -5845.986} C_VEL
LIN {X 0,Y 502.09,Z 632.049,A -85,B 0,C 180,E1 -5847.593,E2 -5847.593} C_VEL
LIN {X 0,Y 501.988,Z 633.391,A -85,B 0,C 180,E1 -5849.197,E2 -5849.197} C_VEL
LIN {X 0,Y 501.988,Z 633.389,A -85,B 0,C 180,E1 -5850.801,E2 -5850.801} C_VEL
LIN {X 0,Y 502.089,Z 632.044,A -85,B 0,C 180,E1 -5852.406,E2 -5852.406} C_VEL
LIN {X 0,Y 502.114,Z 629.323,A -85,B 0,C 180,E1 -5854.012,E2 -5854.012} C_VEL
LIN {X 0,Y 502.198,Z 625.154,A -85,B 0,C 180,E1 -5855.621,E2 -5855.621} C_VEL
LIN {X 0,Y 502.252,Z 619.41,A -85,B 0,C 180,E1 -5857.234,E2 -5857.234} C_VEL
LIN {X 0,Y 502.425,Z 612.94,A -85,B 0,C 180,E1 -5858.648,E2 -5858.648} C_VEL
LIN {X 0,Y 502.678,Z 604.903,A -85,B 0,C 180,E1 -5860.064,E2 -5860.064} C_VEL
LIN {X 0,Y 502.988,Z 596.5,A -85,B 0,C 180,E1 -5861.28,E2 -5861.28} C_VEL
LIN {X 0,Y 503.36,Z 586.746,A -85,B 0,C 180,E1 -5862.457,E2 -5862.457} C_VEL
LIN {X 0,Y 503.768,Z 576.213,A -85,B 0,C 180,E1 -5863.513,E2 -5863.513} C_VEL
LIN {X 0,Y 504.307,Z 563.889,A -85,B 0,C 180,E1 -5864.527,E2 -5864.527} C_VEL
LIN {X 0,Y 504.759,Z 551.673,A -85,B 0,C 180,E1 -5865.339,E2 -5865.339} C_VEL
LIN {X 0,Y 505.276,Z 538.121,A -85,B 0,C 180,E1 -5866.047,E2 -5866.047} C_VEL
LIN {X 0,Y 505.638,Z 524.081,A -85,B 0,C 180,E1 -5866.601,E2 -5866.601} C_VEL
LIN {X 0,Y 505.952,Z 510.051,A -85,B 0,C 180,E1 -5866.985,E2 -5866.985} C_VEL
LIN {X 0,Y 506.191,Z 485.984,A -85,B 0,C 180,E1 -5867.367,E2 -5867.367} C_VEL
LIN {X 0,Y 506.881,Z 385.827,A -85,B 0,C 180,E1 -5868.81,E2 -5868.81} C_VEL
LIN {X 0,Y 504.079,Z 369.443,A -85,B 0,C 180,E1 -5869.167,E2 -5869.167} C_VEL
LIN {X 0,Y 504.778,Z 349.304,A -85,B 0,C 180,E1 -5872.08,E2 -5872.08} C_VEL
LIN {X 0,Y 505.488,Z 329.61,A -85,B 0,C 180,E1 -5874.987,E2 -5874.987} C_VEL
LIN {X 0,Y 503.447,Z 319.116,A -85,B 0,C 180,E1 -5876.693,E2 -5876.693} C_VEL
LIN {X 0,Y 502.866,Z 316.474,A -85,B 0,C 180,E1 -5877.158,E2 -5877.158} C_VEL
LIN {X 0,Y 502.807,Z 316.477,A -85,B 0,C 180,E1 -5880.21,E2 -5880.21} C_VEL
LIN {X 0,Y 502.829,Z 316.478,A -85,B 0,C 180,E1 -5883.03,E2 -5883.03} C_VEL
LIN {X 0,Y 502.78,Z 316.477,A -85,B 0,C 180,E1 -5885.949,E2 -5885.949} C_VEL
LIN {X 0,Y 502.799,Z 316.479,A -85,B 0,C 180,E1 -5888.975,E2 -5888.975} C_VEL
LIN {X 0,Y 502.823,Z 316.474,A -85,B 0,C 180,E1 -5891.064,E2 -5891.064} C_VEL
LIN {X 0,Y 502.797,Z 316.483,A -85,B 0,C 180,E1 -5894.531,E2 -5894.531} C_VEL
LIN {X 0,Y 502.825,Z 316.473,A -85,B 0,C 180,E1 -5897.863,E2 -5897.863} C_VEL
LIN {X 0,Y 502.797,Z 316.476,A -85,B 0,C 180,E1 -5901.023,E2 -5901.023} C_VEL
LIN {X 0,Y 502.778,Z 316.482,A -85,B 0,C 180,E1 -5904.167,E2 -5904.167} C_VEL
LIN {X 0,Y 502.826,Z 316.471,A -85,B 0,C 180,E1 -5906.993,E2 -5906.993} C_VEL
LIN {X 0,Y 502.824,Z 316.476,A -85,B 0,C 180,E1 -5910.061,E2 -5910.061} C_VEL
LIN {X 0,Y 502.829,Z 316.475,A -85,B 0,C 180,E1 -5912.533,E2 -5912.533} C_VEL
LIN {X 0,Y 502.815,Z 316.473,A -85,B 0,C 180,E1 -5915.299,E2 -5915.299} C_VEL
LIN {X 0,Y 502.772,Z 316.479,A -85,B 0,C 180,E1 -5917.826,E2 -5917.826} C_VEL
LIN {X 0,Y 502.817,Z 316.474,A -85,B 0,C 180,E1 -5920.4,E2 -5920.4} C_VEL
LIN {X 0,Y 502.825,Z 316.472,A -85,B 0,C 180,E1 -5922.931,E2 -5922.931} C_VEL
LIN {X 0,Y 502.836,Z 316.468,A -85,B 0,C 180,E1 -5925.429,E2 -5925.429} C_VEL
LIN {X 0,Y 502.867,Z 316.463,A -85,B 0,C 180,E1 -5928.716,E2 -5928.716} C_VEL
LIN {X 0,Y 502.891,Z 316.468,A -85,B 0,C 180,E1 -5931.966,E2 -5931.966} C_VEL
LIN {X 0,Y 502.919,Z 316.462,A -85,B 0,C 180,E1 -5934.386,E2 -5934.386} C_VEL
LIN {X 0,Y 503.004,Z 316.452,A -85,B 0,C 180,E1 -5937.597,E2 -5937.597} C_VEL
LIN {X 0,Y 502.992,Z 316.454,A -85,B 0,C 180,E1 -5940,E2 -5940} C_VEL
LIN {X 0,Y 503.003,Z 316.45,A -85,B 0,C 180,E1 -5942.402,E2 -5942.402} C_VEL
LIN {X 0,Y 502.877,Z 316.47,A -85,B 0,C 180,E1 -5945.614,E2 -5945.614} C_VEL
LIN {X 0,Y 502.838,Z 316.471,A -85,B 0,C 180,E1 -5948.034,E2 -5948.034} C_VEL
LIN {X 0,Y 502.862,Z 316.473,A -85,B 0,C 180,E1 -5951.283,E2 -5951.283} C_VEL
LIN {X 0,Y 502.81,Z 316.474,A -85,B 0,C 180,E1 -5954.572,E2 -5954.572} C_VEL
LIN {X 0,Y 502.79,Z 316.478,A -85,B 0,C 180,E1 -5957.909,E2 -5957.909} C_VEL
LIN {X 0,Y 502.819,Z 316.473,A -85,B 0,C 180,E1 -5960.536,E2 -5960.536} C_VEL
LIN {X 0,Y 502.775,Z 316.482,A -85,B 0,C 180,E1 -5963.041,E2 -5963.041} C_VEL
LIN {X 0,Y 502.824,Z 316.474,A -85,B 0,C 180,E1 -5966.568,E2 -5966.568} C_VEL
LIN {X 0,Y 502.8,Z 316.477,A -85,B 0,C 180,E1 -5969.934,E2 -5969.934} C_VEL
LIN {X 0,Y 502.819,Z 316.476,A -85,B 0,C 180,E1 -5973.032,E2 -5973.032} C_VEL
LIN {X 0,Y 502.763,Z 316.48,A -85,B 0,C 180,E1 -5975.952,E2 -5975.952} C_VEL
LIN {X 0,Y 502.791,Z 316.481,A -85,B 0,C 180,E1 -5978.977,E2 -5978.977} C_VEL
LIN {X 0,Y 502.786,Z 316.476,A -85,B 0,C 180,E1 -5982.14,E2 -5982.14} C_VEL
LIN {X 0,Y 502.777,Z 316.479,A -85,B 0,C 180,E1 -5985.471,E2 -5985.471} C_VEL
LIN {X 0,Y 502.812,Z 316.482,A -85,B 0,C 180,E1 -5988.935,E2 -5988.935} C_VEL
LIN {X 0,Y 502.839,Z 316.653,A -85,B 0,C 180,E1 -5989.466,E2 -5989.466} C_VEL
LIN {X 0,Y 504.315,Z 324.01,A -85,B 0,C 180,E1 -5990.907,E2 -5990.907} C_VEL
LIN {X 0,Y 504.32,Z 330.979,A -85,B 0,C 180,E1 -5992.183,E2 -5992.183} C_VEL
LIN {X 0,Y 504.142,Z 334.982,A -85,B 0,C 180,E1 -5992.902,E2 -5992.902} C_VEL
LIN {X 0,Y 507.032,Z 348.442,A -85,B 0,C 180,E1 -5993.221,E2 -5993.221} C_VEL
LIN {X 0,Y 506.97,Z 358.262,A -85,B 0,C 180,E1 -5993.364,E2 -5993.364} C_VEL
LIN {X 0,Y 506.267,Z 364.111,A -85,B 0,C 180,E1 -5993.423,E2 -5993.423} C_VEL
LIN {X 0,Y 500.667,Z 383.143,A -85,B 0,C 180,E1 -5993.485,E2 -5993.485} C_VEL
LIN {X 0,Y 500.029,Z 388.989,A -85,B 0,C 180,E1 -5993.547,E2 -5993.547} C_VEL
LIN {X 0,Y 499.378,Z 471.606,A -85,B 0,C 180,E1 -5994.777,E2 -5994.777} C_VEL
LIN {X 0,Y 499.075,Z 486.318,A -85,B 0,C 180,E1 -5995.167,E2 -5995.167} C_VEL
LIN {X 0,Y 498.723,Z 499.817,A -85,B 0,C 180,E1 -5995.691,E2 -5995.691} C_VEL
LIN {X 0,Y 498.215,Z 513.842,A -85,B 0,C 180,E1 -5996.419,E2 -5996.419} C_VEL
LIN {X 0,Y 497.656,Z 527.101,A -85,B 0,C 180,E1 -5997.306,E2 -5997.306} C_VEL
LIN {X 0,Y 497.146,Z 539.1,A -85,B 0,C 180,E1 -5998.311,E2 -5998.311} C_VEL
LIN {X 0,Y 496.632,Z 549.521,A -85,B 0,C 180,E1 -5999.374,E2 -5999.374} C_VEL
LIN {X 0,Y 496.253,Z 558.86,A -85,B 0,C 180,E1 -6000.52,E2 -6000.52} C_VEL
LIN {X 0,Y 495.877,Z 567.502,A -85,B 0,C 180,E1 -6001.796,E2 -6001.796} C_VEL
LIN {X 0,Y 495.582,Z 574.38,A -85,B 0,C 180,E1 -6003.013,E2 -6003.013} C_VEL
LIN {X 0,Y 495.333,Z 580.629,A -85,B 0,C 180,E1 -6004.359,E2 -6004.359} C_VEL
LIN {X 0,Y 495.211,Z 585.623,A -85,B 0,C 180,E1 -6005.698,E2 -6005.698} C_VEL
LIN {X 0,Y 495.049,Z 590.32,A -85,B 0,C 180,E1 -6007.334,E2 -6007.334} C_VEL
LIN {X 0,Y 494.969,Z 592.427,A -85,B 0,C 180,E1 -6008.337,E2 -6008.337} C_VEL
LIN {X 0,Y 494.933,Z 594.871,A -85,B 0,C 180,E1 -6010.075,E2 -6010.075} C_VEL
LIN {X 0,Y 494.942,Z 595.813,A -85,B 0,C 180,E1 -6011.798,E2 -6011.798} C_VEL
LIN {X 0,Y 494.883,Z 595.314,A -85,B 0,C 180,E1 -6013.5,E2 -6013.5} C_VEL
LIN {X 0,Y 494.992,Z 593.383,A -85,B 0,C 180,E1 -6015.194,E2 -6015.194} C_VEL
LIN {X 0,Y 495.052,Z 589.988,A -85,B 0,C 180,E1 -6016.872,E2 -6016.872} C_VEL
LIN {X 0,Y 495.211,Z 585.074,A -85,B 0,C 180,E1 -6018.541,E2 -6018.541} C_VEL
LIN {X 0,Y 495.336,Z 580.346,A -85,B 0,C 180,E1 -6019.785,E2 -6019.785} C_VEL
LIN {X 0,Y 495.565,Z 573.497,A -85,B 0,C 180,E1 -6021.232,E2 -6021.232} C_VEL
LIN {X 0,Y 495.935,Z 565.017,A -85,B 0,C 180,E1 -6022.673,E2 -6022.673} C_VEL
LIN {X 0,Y 496.338,Z 556.195,A -85,B 0,C 180,E1 -6023.905,E2 -6023.905} C_VEL
LIN {X 0,Y 496.802,Z 545.559,A -85,B 0,C 180,E1 -6025.132,E2 -6025.132} C_VEL
LIN {X 0,Y 497.258,Z 534.832,A -85,B 0,C 180,E1 -6026.151,E2 -6026.151} C_VEL
LIN {X 0,Y 497.818,Z 523.082,A -85,B 0,C 180,E1 -6027.067,E2 -6027.067} C_VEL
LIN {X 0,Y 498.343,Z 510.155,A -85,B 0,C 180,E1 -6027.879,E2 -6027.879} C_VEL
LIN {X 0,Y 498.78,Z 497.532,A -85,B 0,C 180,E1 -6028.497,E2 -6028.497} C_VEL
LIN {X 0,Y 499.107,Z 483.347,A -85,B 0,C 180,E1 -6029.012,E2 -6029.012} C_VEL
LIN {X 0,Y 499.386,Z 469.555,A -85,B 0,C 180,E1 -6029.346,E2 -6029.346} C_VEL
LIN {X 0,Y 500.227,Z 348.918,A -85,B 0,C 180,E1 -6031.124,E2 -6031.124} C_VEL
LIN {X 0,Y 497.229,Z 335.031,A -85,B 0,C 180,E1 -6031.461,E2 -6031.461} C_VEL
LIN {X 0,Y 497.548,Z 326.371,A -85,B 0,C 180,E1 -6033.037,E2 -6033.037} C_VEL
LIN {X 0,Y 495.815,Z 317.352,A -85,B 0,C 180,E1 -6034.829,E2 -6034.829} C_VEL
LIN {X 0,Y 495.875,Z 317.344,A -85,B 0,C 180,E1 -6037.329,E2 -6037.329} C_VEL
LIN {X 0,Y 495.781,Z 317.355,A -85,B 0,C 180,E1 -6039.795,E2 -6039.795} C_VEL
LIN {X 0,Y 495.785,Z 317.348,A -85,B 0,C 180,E1 -6042.277,E2 -6042.277} C_VEL
LIN {X 0,Y 495.805,Z 317.349,A -85,B 0,C 180,E1 -6045.625,E2 -6045.625} C_VEL
LIN {X 0,Y 495.777,Z 317.355,A -85,B 0,C 180,E1 -6049.029,E2 -6049.029} C_VEL
LIN {X 0,Y 495.739,Z 317.356,A -85,B 0,C 180,E1 -6051.63,E2 -6051.63} C_VEL
LIN {X 0,Y 495.71,Z 317.358,A -85,B 0,C 180,E1 -6054.278,E2 -6054.278} C_VEL
LIN {X 0,Y 495.727,Z 317.363,A -85,B 0,C 180,E1 -6056.98,E2 -6056.98} C_VEL
LIN {X 0,Y 495.736,Z 317.354,A -85,B 0,C 180,E1 -6060.142,E2 -6060.142} C_VEL
LIN {X 0,Y 495.726,Z 317.36,A -85,B 0,C 180,E1 -6063.233,E2 -6063.233} C_VEL
LIN {X 0,Y 495.726,Z 317.356,A -85,B 0,C 180,E1 -6065.54,E2 -6065.54} C_VEL
LIN {X 0,Y 495.732,Z 317.362,A -85,B 0,C 180,E1 -6068.764,E2 -6068.764} C_VEL
LIN {X 0,Y 495.722,Z 317.356,A -85,B 0,C 180,E1 -6071.785,E2 -6071.785} C_VEL
LIN {X 0,Y 495.73,Z 317.358,A -85,B 0,C 180,E1 -6075.142,E2 -6075.142} C_VEL
LIN {X 0,Y 495.721,Z 317.358,A -85,B 0,C 180,E1 -6078.216,E2 -6078.216} C_VEL
LIN {X 0,Y 495.711,Z 317.358,A -85,B 0,C 180,E1 -6081.405,E2 -6081.405} C_VEL
LIN {X 0,Y 495.727,Z 317.362,A -85,B 0,C 180,E1 -6084.461,E2 -6084.461} C_VEL
LIN {X 0,Y 495.75,Z 317.352,A -85,B 0,C 180,E1 -6087.405,E2 -6087.405} C_VEL
LIN {X 0,Y 495.738,Z 317.359,A -85,B 0,C 180,E1 -6090.252,E2 -6090.252} C_VEL
LIN {X 0,Y 495.738,Z 317.354,A -85,B 0,C 180,E1 -6093.271,E2 -6093.271} C_VEL
LIN {X 0,Y 495.71,Z 317.358,A -85,B 0,C 180,E1 -6095.723,E2 -6095.723} C_VEL
LIN {X 0,Y 495.735,Z 317.363,A -85,B 0,C 180,E1 -6098.371,E2 -6098.371} C_VEL
LIN {X 0,Y 495.768,Z 317.351,A -85,B 0,C 180,E1 -6100.971,E2 -6100.971} C_VEL
LIN {X 0,Y 495.804,Z 317.35,A -85,B 0,C 180,E1 -6104.558,E2 -6104.558} C_VEL
LIN {X 0,Y 495.831,Z 317.348,A -85,B 0,C 180,E1 -6107.966,E2 -6107.966} C_VEL
LIN {X 0,Y 495.834,Z 317.342,A -85,B 0,C 180,E1 -6111.03,E2 -6111.03} C_VEL
LIN {X 0,Y 495.88,Z 317.342,A -85,B 0,C 180,E1 -6114.307,E2 -6114.307} C_VEL
LIN {X 0,Y 495.988,Z 317.325,A -85,B 0,C 180,E1 -6117.564,E2 -6117.564} C_VEL
LIN {X 0,Y 495.964,Z 317.326,A -85,B 0,C 180,E1 -6120.812,E2 -6120.812} C_VEL
LIN {X 0,Y 495.988,Z 317.325,A -85,B 0,C 180,E1 -6122.437,E2 -6122.437} C_VEL
LIN {X 0,Y 495.883,Z 317.341,A -85,B 0,C 180,E1 -6125.694,E2 -6125.694} C_VEL
LIN {X 0,Y 495.841,Z 317.341,A -85,B 0,C 180,E1 -6128.97,E2 -6128.97} C_VEL
LIN {X 0,Y 495.832,Z 317.347,A -85,B 0,C 180,E1 -6132.035,E2 -6132.035} C_VEL
LIN {X 0,Y 495.828,Z 317.347,A -85,B 0,C 180,E1 -6135.452,E2 -6135.452} C_VEL
LIN {X 0,Y 495.811,Z 317.346,A -85,B 0,C 180,E1 -6138.247,E2 -6138.247} C_VEL
LIN {X 0,Y 495.778,Z 317.349,A -85,B 0,C 180,E1 -6140.756,E2 -6140.756} C_VEL
LIN {X 0,Y 495.746,Z 317.358,A -85,B 0,C 180,E1 -6143.388,E2 -6143.388} C_VEL
LIN {X 0,Y 495.827,Z 317.343,A -85,B 0,C 180,E1 -6146.749,E2 -6146.749} C_VEL
LIN {X 0,Y 495.77,Z 317.355,A -85,B 0,C 180,E1 -6149.746,E2 -6149.746} C_VEL
LIN {X 0,Y 495.771,Z 317.35,A -85,B 0,C 180,E1 -6152.594,E2 -6152.594} C_VEL
LIN {X 0,Y 495.749,Z 317.359,A -85,B 0,C 180,E1 -6155.538,E2 -6155.538} C_VEL
LIN {X 0,Y 495.766,Z 317.352,A -85,B 0,C 180,E1 -6158.768,E2 -6158.768} C_VEL
LIN {X 0,Y 495.76,Z 317.353,A -85,B 0,C 180,E1 -6161.781,E2 -6161.781} C_VEL
LIN {X 0,Y 495.753,Z 317.359,A -85,B 0,C 180,E1 -6165.139,E2 -6165.139} C_VEL
LIN {X 0,Y 495.76,Z 317.351,A -85,B 0,C 180,E1 -6168.219,E2 -6168.219} C_VEL
LIN {X 0,Y 495.755,Z 317.356,A -85,B 0,C 180,E1 -6171.408,E2 -6171.408} C_VEL
LIN {X 0,Y 495.753,Z 317.353,A -85,B 0,C 180,E1 -6174.462,E2 -6174.462} C_VEL
LIN {X 0,Y 495.771,Z 317.356,A -85,B 0,C 180,E1 -6177.405,E2 -6177.405} C_VEL
LIN {X 0,Y 495.769,Z 317.356,A -85,B 0,C 180,E1 -6180.253,E2 -6180.253} C_VEL
LIN {X 0,Y 495.837,Z 317.518,A -85,B 0,C 180,E1 -6182.684,E2 -6182.684} C_VEL
LIN {X 0,Y 498.562,Z 330.602,A -85,B 0,C 180,E1 -6184.83,E2 -6184.83} C_VEL
LIN {X 0,Y 498.045,Z 346.232,A -85,B 0,C 180,E1 -6187.166,E2 -6187.166} C_VEL
LIN {X 0,Y 497.285,Z 366.691,A -85,B 0,C 180,E1 -6190.172,E2 -6190.172} C_VEL
LIN {X 0,Y 497.238,Z 369.696,A -85,B 0,C 180,E1 -6190.576,E2 -6190.576} C_VEL
LIN {X 0,Y 500.171,Z 387.161,A -85,B 0,C 180,E1 -6190.951,E2 -6190.951} C_VEL
LIN {X 0,Y 499.247,Z 507.519,A -85,B 0,C 180,E1 -6192.725,E2 -6192.725} C_VEL
LIN {X 0,Y 498.863,Z 522.214,A -85,B 0,C 180,E1 -6193.108,E2 -6193.108} C_VEL
LIN {X 0,Y 498.48,Z 535.651,A -85,B 0,C 180,E1 -6193.621,E2 -6193.621} C_VEL
LIN {X 0,Y 497.981,Z 549.687,A -85,B 0,C 180,E1 -6194.34,E2 -6194.34} C_VEL
LIN {X 0,Y 497.406,Z 562.238,A -85,B 0,C 180,E1 -6195.161,E2 -6195.161} C_VEL
LIN {X 0,Y 496.876,Z 574.889,A -85,B 0,C 180,E1 -6196.19,E2 -6196.19} C_VEL
LIN {X 0,Y 496.404,Z 586.167,A -85,B 0,C 180,E1 -6197.323,E2 -6197.323} C_VEL
LIN {X 0,Y 495.972,Z 596.274,A -85,B 0,C 180,E1 -6198.557,E2 -6198.557} C_VEL
LIN {X 0,Y 495.615,Z 604.671,A -85,B 0,C 180,E1 -6199.789,E2 -6199.789} C_VEL
LIN {X 0,Y 495.365,Z 612.702,A -85,B 0,C 180,E1 -6201.227,E2 -6201.227} C_VEL
LIN {X 0,Y 495.174,Z 619.169,A -85,B 0,C 180,E1 -6202.66,E2 -6202.66} C_VEL
LIN {X 0,Y 495.109,Z 624.905,A -85,B 0,C 180,E1 -6204.297,E2 -6204.297} C_VEL
LIN {X 0,Y 495.011,Z 629.064,A -85,B 0,C 180,E1 -6205.929,E2 -6205.929} C_VEL
LIN {X 0,Y 494.996,Z 631.781,A -85,B 0,C 180,E1 -6207.558,E2 -6207.558} C_VEL
LIN {X 0,Y 494.908,Z 633.123,A -85,B 0,C 180,E1 -6209.186,E2 -6209.186} C_VEL
LIN {X 0,Y 494.908,Z 633.12,A -85,B 0,C 180,E1 -6210.813,E2 -6210.813} C_VEL
LIN {X 0,Y 494.996,Z 631.773,A -85,B 0,C 180,E1 -6212.44,E2 -6212.44} C_VEL
LIN {X 0,Y 495.011,Z 629.05,A -85,B 0,C 180,E1 -6214.07,E2 -6214.07} C_VEL
LIN {X 0,Y 495.114,Z 624.879,A -85,B 0,C 180,E1 -6215.702,E2 -6215.702} C_VEL
LIN {X 0,Y 495.173,Z 619.132,A -85,B 0,C 180,E1 -6217.338,E2 -6217.338} C_VEL
LIN {X 0,Y 495.363,Z 612.658,A -85,B 0,C 180,E1 -6218.772,E2 -6218.772} C_VEL
LIN {X 0,Y 495.616,Z 604.617,A -85,B 0,C 180,E1 -6220.209,E2 -6220.209} C_VEL
LIN {X 0,Y 495.946,Z 596.21,A -85,B 0,C 180,E1 -6221.442,E2 -6221.442} C_VEL
LIN {X 0,Y 496.402,Z 586.094,A -85,B 0,C 180,E1 -6222.676,E2 -6222.676} C_VEL
LIN {X 0,Y 496.865,Z 574.805,A -85,B 0,C 180,E1 -6223.808,E2 -6223.808} C_VEL
LIN {X 0,Y 497.411,Z 562.15,A -85,B 0,C 180,E1 -6224.837,E2 -6224.837} C_VEL
LIN {X 0,Y 497.949,Z 549.587,A -85,B 0,C 180,E1 -6225.659,E2 -6225.659} C_VEL
LIN {X 0,Y 498.464,Z 536.672,A -85,B 0,C 180,E1 -6226.325,E2 -6226.325} C_VEL
LIN {X 0,Y 498.828,Z 523.024,A -85,B 0,C 180,E1 -6226.86,E2 -6226.86} C_VEL
LIN {X 0,Y 499.207,Z 508.615,A -85,B 0,C 180,E1 -6227.248,E2 -6227.248} C_VEL
LIN {X 0,Y 499.617,Z 467.932,A -85,B 0,C 180,E1 -6227.867,E2 -6227.867} C_VEL
LIN {X 0,Y 500.08,Z 386.099,A -85,B 0,C 180,E1 -6229.07,E2 -6229.07} C_VEL
LIN {X 0,Y 497.163,Z 369.179,A -85,B 0,C 180,E1 -6229.444,E2 -6229.444} C_VEL
LIN {X 0,Y 497.859,Z 350.545,A -85,B 0,C 180,E1 -6232.185,E2 -6232.185} C_VEL
LIN {X 0,Y 498.64,Z 331.665,A -85,B 0,C 180,E1 -6235.012,E2 -6235.012} C_VEL
LIN {X 0,Y 497.031,Z 322.93,A -85,B 0,C 180,E1 -6236.448,E2 -6236.448} C_VEL
LIN {X 0,Y 495.813,Z 317.351,A -85,B 0,C 180,E1 -6237.43,E2 -6237.43} C_VEL
LIN {X 0,Y 495.75,Z 317.359,A -85,B 0,C 180,E1 -6240.686,E2 -6240.686} C_VEL
LIN {X 0,Y 495.758,Z 317.352,A -85,B 0,C 180,E1 -6243.563,E2 -6243.563} C_VEL
LIN {X 0,Y 495.731,Z 317.358,A -85,B 0,C 180,E1 -6246.542,E2 -6246.542} C_VEL
LIN {X 0,Y 495.772,Z 317.352,A -85,B 0,C 180,E1 -6249.635,E2 -6249.635} C_VEL
LIN {X 0,Y 495.733,Z 317.357,A -85,B 0,C 180,E1 -6252.506,E2 -6252.506} C_VEL
LIN {X 0,Y 495.745,Z 317.352,A -85,B 0,C 180,E1 -6255.138,E2 -6255.138} C_VEL
LIN {X 0,Y 495.772,Z 317.354,A -85,B 0,C 180,E1 -6258.22,E2 -6258.22} C_VEL
LIN {X 0,Y 495.745,Z 317.352,A -85,B 0,C 180,E1 -6261.408,E2 -6261.408} C_VEL
LIN {X 0,Y 495.75,Z 317.359,A -85,B 0,C 180,E1 -6264.462,E2 -6264.462} C_VEL
LIN {X 0,Y 495.762,Z 317.35,A -85,B 0,C 180,E1 -6267.405,E2 -6267.405} C_VEL
LIN {X 0,Y 495.775,Z 317.355,A -85,B 0,C 180,E1 -6270.254,E2 -6270.254} C_VEL
LIN {X 0,Y 495.827,Z 317.341,A -85,B 0,C 180,E1 -6273.248,E2 -6273.248} C_VEL
LIN {X 0,Y 495.735,Z 317.357,A -85,B 0,C 180,E1 -6275.724,E2 -6275.724} C_VEL
LIN {X 0,Y 495.735,Z 317.361,A -85,B 0,C 180,E1 -6278.37,E2 -6278.37} C_VEL
LIN {X 0,Y 495.776,Z 317.347,A -85,B 0,C 180,E1 -6280.971,E2 -6280.971} C_VEL
LIN {X 0,Y 495.77,Z 317.353,A -85,B 0,C 180,E1 -6283.529,E2 -6283.529} C_VEL
LIN {X 0,Y 495.784,Z 317.355,A -85,B 0,C 180,E1 -6286.055,E2 -6286.055} C_VEL
LIN {X 0,Y 495.842,Z 317.339,A -85,B 0,C 180,E1 -6288.554,E2 -6288.554} C_VEL
LIN {X 0,Y 495.862,Z 317.346,A -85,B 0,C 180,E1 -6291.852,E2 -6291.852} C_VEL
LIN {X 0,Y 495.876,Z 317.34,A -85,B 0,C 180,E1 -6294.306,E2 -6294.306} C_VEL
LIN {X 0,Y 495.972,Z 317.328,A -85,B 0,C 180,E1 -6297.563,E2 -6297.563} C_VEL
LIN {X 0,Y 495.961,Z 317.33,A -85,B 0,C 180,E1 -6300,E2 -6300} C_VEL
LIN {X 0,Y 495.971,Z 317.326,A -85,B 0,C 180,E1 -6302.436,E2 -6302.436} C_VEL
LIN {X 0,Y 495.834,Z 317.347,A -85,B 0,C 180,E1 -6305.694,E2 -6305.694} C_VEL
LIN {X 0,Y 495.801,Z 317.346,A -85,B 0,C 180,E1 -6308.149,E2 -6308.149} C_VEL
LIN {X 0,Y 495.838,Z 317.35,A -85,B 0,C 180,E1 -6311.445,E2 -6311.445} C_VEL
LIN {X 0,Y 495.762,Z 317.353,A -85,B 0,C 180,E1 -6314.783,E2 -6314.783} C_VEL
LIN {X 0,Y 495.761,Z 317.352,A -85,B 0,C 180,E1 -6318.235,E2 -6318.235} C_VEL
LIN {X 0,Y 495.764,Z 317.353,A -85,B 0,C 180,E1 -6320.756,E2 -6320.756} C_VEL
LIN {X 0,Y 495.728,Z 317.363,A -85,B 0,C 180,E1 -6323.388,E2 -6323.388} C_VEL
LIN {X 0,Y 495.763,Z 317.356,A -85,B 0,C 180,E1 -6326.738,E2 -6326.738} C_VEL
LIN {X 0,Y 495.748,Z 317.355,A -85,B 0,C 180,E1 -6330.146,E2 -6330.146} C_VEL
LIN {X 0,Y 495.779,Z 317.353,A -85,B 0,C 180,E1 -6333.244,E2 -6333.244} C_VEL
LIN {X 0,Y 495.71,Z 317.359,A -85,B 0,C 180,E1 -6336.089,E2 -6336.089} C_VEL
LIN {X 0,Y 495.753,Z 317.36,A -85,B 0,C 180,E1 -6338.768,E2 -6338.768} C_VEL
LIN {X 0,Y 495.747,Z 317.353,A -85,B 0,C 180,E1 -6341.782,E2 -6341.782} C_VEL
LIN {X 0,Y 495.728,Z 317.36,A -85,B 0,C 180,E1 -6345.141,E2 -6345.141} C_VEL
LIN {X 0,Y 495.748,Z 317.36,A -85,B 0,C 180,E1 -6348.219,E2 -6348.219} C_VEL
LIN {X 0,Y 495.758,Z 317.439,A -85,B 0,C 180,E1 -6349.214,E2 -6349.214} C_VEL
LIN {X 0,Y 497.484,Z 326.353,A -85,B 0,C 180,E1 -6350.985,E2 -6350.985} C_VEL
LIN {X 0,Y 497.253,Z 335.219,A -85,B 0,C 180,E1 -6352.617,E2 -6352.617} C_VEL
LIN {X 0,Y 500.258,Z 348.702,A -85,B 0,C 180,E1 -6352.953,E2 -6352.953} C_VEL
LIN {X 0,Y 500.029,Z 388.989,A -85,B 0,C 180,E1 -6353.547,E2 -6353.547} C_VEL
LIN {X 0,Y 499.396,Z 394.833,A -85,B 0,C 180,E1 -6353.61,E2 -6353.61} C_VEL
LIN {X 0,Y 493.796,Z 413.859,A -85,B 0,C 180,E1 -6353.676,E2 -6353.676} C_VEL
LIN {X 0,Y 493.064,Z 419.707,A -85,B 0,C 180,E1 -6353.735,E2 -6353.735} C_VEL
LIN {X 0,Y 492.598,Z 472.31,A -85,B 0,C 180,E1 -6354.539,E2 -6354.539} C_VEL
LIN {X 0,Y 492.263,Z 487.137,A -85,B 0,C 180,E1 -6354.943,E2 -6354.943} C_VEL
LIN {X 0,Y 491.926,Z 500.182,A -85,B 0,C 180,E1 -6355.46,E2 -6355.46} C_VEL
LIN {X 0,Y 491.452,Z 512.587,A -85,B 0,C 180,E1 -6356.103,E2 -6356.103} C_VEL
LIN {X 0,Y 490.903,Z 525.037,A -85,B 0,C 180,E1 -6356.921,E2 -6356.921} C_VEL
LIN {X 0,Y 490.366,Z 536.141,A -85,B 0,C 180,E1 -6357.819,E2 -6357.819} C_VEL
LIN {X 0,Y 489.881,Z 547.176,A -85,B 0,C 180,E1 -6358.906,E2 -6358.906} C_VEL
LIN {X 0,Y 489.376,Z 556.933,A -85,B 0,C 180,E1 -6360.064,E2 -6360.064} C_VEL
LIN {X 0,Y 488.915,Z 566.674,A -85,B 0,C 180,E1 -6361.468,E2 -6361.468} C_VEL
LIN {X 0,Y 488.554,Z 574.742,A -85,B 0,C 180,E1 -6362.901,E2 -6362.901} C_VEL
LIN {X 0,Y 488.262,Z 581.581,A -85,B 0,C 180,E1 -6364.418,E2 -6364.418} C_VEL
LIN {X 0,Y 488.12,Z 586.463,A -85,B 0,C 180,E1 -6365.775,E2 -6365.775} C_VEL
LIN {X 0,Y 487.973,Z 590.379,A -85,B 0,C 180,E1 -6367.183,E2 -6367.183} C_VEL
LIN {X 0,Y 487.861,Z 593.741,A -85,B 0,C 180,E1 -6368.892,E2 -6368.892} C_VEL
LIN {X 0,Y 487.824,Z 595.639,A -85,B 0,C 180,E1 -6370.65,E2 -6370.65} C_VEL
LIN {X 0,Y 487.836,Z 596.061,A -85,B 0,C 180,E1 -6372.391,E2 -6372.391} C_VEL
LIN {X 0,Y 487.785,Z 595.058,A -85,B 0,C 180,E1 -6374.113,E2 -6374.113} C_VEL
LIN {X 0,Y 487.915,Z 592.63,A -85,B 0,C 180,E1 -6375.827,E2 -6375.827} C_VEL
LIN {X 0,Y 488.024,Z 588.761,A -85,B 0,C 180,E1 -6377.526,E2 -6377.526} C_VEL
LIN {X 0,Y 488.158,Z 584.796,A -85,B 0,C 180,E1 -6378.794,E2 -6378.794} C_VEL
LIN {X 0,Y 488.299,Z 579.925,A -85,B 0,C 180,E1 -6380.055,E2 -6380.055} C_VEL
LIN {X 0,Y 488.584,Z 572.914,A -85,B 0,C 180,E1 -6381.522,E2 -6381.522} C_VEL
LIN {X 0,Y 488.951,Z 564.731,A -85,B 0,C 180,E1 -6382.911,E2 -6382.911} C_VEL
LIN {X 0,Y 489.403,Z 555.238,A -85,B 0,C 180,E1 -6384.232,E2 -6384.232} C_VEL
LIN {X 0,Y 489.965,Z 544.331,A -85,B 0,C 180,E1 -6385.476,E2 -6385.476} C_VEL
LIN {X 0,Y 490.474,Z 533.269,A -85,B 0,C 180,E1 -6386.509,E2 -6386.509} C_VEL
LIN {X 0,Y 491.037,Z 521.065,A -85,B 0,C 180,E1 -6387.437,E2 -6387.437} C_VEL
LIN {X 0,Y 491.571,Z 509.342,A -85,B 0,C 180,E1 -6388.157,E2 -6388.157} C_VEL
LIN {X 0,Y 492.033,Z 495.626,A -85,B 0,C 180,E1 -6388.814,E2 -6388.814} C_VEL
LIN {X 0,Y 492.363,Z 481.722,A -85,B 0,C 180,E1 -6389.301,E2 -6389.301} C_VEL
LIN {X 0,Y 492.641,Z 467.423,A -85,B 0,C 180,E1 -6389.627,E2 -6389.627} C_VEL
LIN {X 0,Y 493.46,Z 349.592,A -85,B 0,C 180,E1 -6391.385,E2 -6391.385} C_VEL
LIN {X 0,Y 490.355,Z 335.245,A -85,B 0,C 180,E1 -6391.746,E2 -6391.746} C_VEL
LIN {X 0,Y 490.466,Z 326.925,A -85,B 0,C 180,E1 -6393.287,E2 -6393.287} C_VEL
LIN {X 0,Y 488.784,Z 318.228,A -85,B 0,C 180,E1 -6395.027,E2 -6395.027} C_VEL
LIN {X 0,Y 488.819,Z 318.223,A -85,B 0,C 180,E1 -6397.435,E2 -6397.435} C_VEL
LIN {X 0,Y 488.75,Z 318.229,A -85,B 0,C 180,E1 -6399.937,E2 -6399.937} C_VEL
LIN {X 0,Y 488.736,Z 318.226,A -85,B 0,C 180,E1 -6402.457,E2 -6402.457} C_VEL
LIN {X 0,Y 488.758,Z 318.225,A -85,B 0,C 180,E1 -6405.856,E2 -6405.856} C_VEL
LIN {X 0,Y 488.737,Z 318.233,A -85,B 0,C 180,E1 -6409.314,E2 -6409.314} C_VEL
LIN {X 0,Y 488.695,Z 318.231,A -85,B 0,C 180,E1 -6411.958,E2 -6411.958} C_VEL
LIN {X 0,Y 488.696,Z 318.239,A -85,B 0,C 180,E1 -6415.041,E2 -6415.041} C_VEL
LIN {X 0,Y 488.68,Z 318.237,A -85,B 0,C 180,E1 -6417.401,E2 -6417.401} C_VEL
LIN {X 0,Y 488.681,Z 318.234,A -85,B 0,C 180,E1 -6420.358,E2 -6420.358} C_VEL
LIN {X 0,Y 488.691,Z 318.233,A -85,B 0,C 180,E1 -6423.477,E2 -6423.477} C_VEL
LIN {X 0,Y 488.646,Z 318.239,A -85,B 0,C 180,E1 -6426.349,E2 -6426.349} C_VEL
LIN {X 0,Y 488.682,Z 318.236,A -85,B 0,C 180,E1 -6429.257,E2 -6429.257} C_VEL
LIN {X 0,Y 488.665,Z 318.235,A -85,B 0,C 180,E1 -6431.595,E2 -6431.595} C_VEL
LIN {X 0,Y 488.694,Z 318.239,A -85,B 0,C 180,E1 -6434.804,E2 -6434.804} C_VEL
LIN {X 0,Y 488.646,Z 318.238,A -85,B 0,C 180,E1 -6437.47,E2 -6437.47} C_VEL
LIN {X 0,Y 488.669,Z 318.242,A -85,B 0,C 180,E1 -6440.743,E2 -6440.743} C_VEL
LIN {X 0,Y 488.643,Z 318.238,A -85,B 0,C 180,E1 -6443.865,E2 -6443.865} C_VEL
LIN {X 0,Y 488.71,Z 318.238,A -85,B 0,C 180,E1 -6446.521,E2 -6446.521} C_VEL
LIN {X 0,Y 488.703,Z 318.231,A -85,B 0,C 180,E1 -6449.78,E2 -6449.78} C_VEL
LIN {X 0,Y 488.697,Z 318.232,A -85,B 0,C 180,E1 -6453.079,E2 -6453.079} C_VEL
LIN {X 0,Y 488.695,Z 318.231,A -85,B 0,C 180,E1 -6455.352,E2 -6455.352} C_VEL
LIN {X 0,Y 488.689,Z 318.236,A -85,B 0,C 180,E1 -6458.043,E2 -6458.043} C_VEL
LIN {X 0,Y 488.731,Z 318.23,A -85,B 0,C 180,E1 -6460.687,E2 -6460.687} C_VEL
LIN {X 0,Y 488.673,Z 318.234,A -85,B 0,C 180,E1 -6463.284,E2 -6463.284} C_VEL
LIN {X 0,Y 488.725,Z 318.231,A -85,B 0,C 180,E1 -6465.85,E2 -6465.85} C_VEL
LIN {X 0,Y 488.807,Z 318.223,A -85,B 0,C 180,E1 -6468.388,E2 -6468.388} C_VEL
LIN {X 0,Y 488.781,Z 318.224,A -85,B 0,C 180,E1 -6471.733,E2 -6471.733} C_VEL
LIN {X 0,Y 488.837,Z 318.22,A -85,B 0,C 180,E1 -6474.224,E2 -6474.224} C_VEL
LIN {X 0,Y 488.955,Z 318.201,A -85,B 0,C 180,E1 -6477.529,E2 -6477.529} C_VEL
LIN {X 0,Y 488.916,Z 318.204,A -85,B 0,C 180,E1 -6480.824,E2 -6480.824} C_VEL
LIN {X 0,Y 488.954,Z 318.201,A -85,B 0,C 180,E1 -6482.472,E2 -6482.472} C_VEL
LIN {X 0,Y 488.841,Z 318.22,A -85,B 0,C 180,E1 -6485.776,E2 -6485.776} C_VEL
LIN {X 0,Y 488.819,Z 318.219,A -85,B 0,C 180,E1 -6488.267,E2 -6488.267} C_VEL
LIN {X 0,Y 488.809,Z 318.223,A -85,B 0,C 180,E1 -6491.613,E2 -6491.613} C_VEL
LIN {X 0,Y 488.765,Z 318.223,A -85,B 0,C 180,E1 -6495.001,E2 -6495.001} C_VEL
LIN {X 0,Y 488.759,Z 318.224,A -85,B 0,C 180,E1 -6498.442,E2 -6498.442} C_VEL
LIN {X 0,Y 488.711,Z 318.231,A -85,B 0,C 180,E1 -6501.071,E2 -6501.071} C_VEL
LIN {X 0,Y 488.683,Z 318.239,A -85,B 0,C 180,E1 -6503.746,E2 -6503.746} C_VEL
LIN {X 0,Y 488.795,Z 318.22,A -85,B 0,C 180,E1 -6506.943,E2 -6506.943} C_VEL
LIN {X 0,Y 488.713,Z 318.229,A -85,B 0,C 180,E1 -6510.363,E2 -6510.363} C_VEL
LIN {X 0,Y 488.738,Z 318.234,A -85,B 0,C 180,E1 -6513.484,E2 -6513.484} C_VEL
LIN {X 0,Y 488.677,Z 318.233,A -85,B 0,C 180,E1 -6516.353,E2 -6516.353} C_VEL
LIN {X 0,Y 488.704,Z 318.238,A -85,B 0,C 180,E1 -6519.254,E2 -6519.254} C_VEL
LIN {X 0,Y 488.711,Z 318.233,A -85,B 0,C 180,E1 -6521.6,E2 -6521.6} C_VEL
LIN {X 0,Y 488.716,Z 318.231,A -85,B 0,C 180,E1 -6524.801,E2 -6524.801} C_VEL
LIN {X 0,Y 488.695,Z 318.236,A -85,B 0,C 180,E1 -6527.474,E2 -6527.474} C_VEL
LIN {X 0,Y 488.737,Z 318.228,A -85,B 0,C 180,E1 -6529.676,E2 -6529.676} C_VEL
LIN {X 0,Y 488.683,Z 318.237,A -85,B 0,C 180,E1 -6532.841,E2 -6532.841} C_VEL
LIN {X 0,Y 488.735,Z 318.226,A -85,B 0,C 180,E1 -6535.887,E2 -6535.887} C_VEL
LIN {X 0,Y 488.695,Z 318.241,A -85,B 0,C 180,E1 -6538.82,E2 -6538.82} C_VEL
LIN {X 0,Y 488.752,Z 318.233,A -85,B 0,C 180,E1 -6542.138,E2 -6542.138} C_VEL
LIN {X 0,Y 488.785,Z 318.273,A -85,B 0,C 180,E1 -6542.431,E2 -6542.431} C_VEL
LIN {X 0,Y 491.555,Z 331.273,A -85,B 0,C 180,E1 -6544.6,E2 -6544.6} C_VEL
LIN {X 0,Y 491.51,Z 338.762,A -85,B 0,C 180,E1 -6545.749,E2 -6545.749} C_VEL
LIN {X 0,Y 490.592,Z 360.556,A -85,B 0,C 180,E1 -6549.013,E2 -6549.013} C_VEL
LIN {X 0,Y 490.291,Z 369.15,A -85,B 0,C 180,E1 -6550.291,E2 -6550.291} C_VEL
LIN {X 0,Y 493.444,Z 388.707,A -85,B 0,C 180,E1 -6550.714,E2 -6550.714} C_VEL
LIN {X 0,Y 492.464,Z 507.025,A -85,B 0,C 180,E1 -6552.48,E2 -6552.48} C_VEL
LIN {X 0,Y 492.049,Z 521.886,A -85,B 0,C 180,E1 -6552.869,E2 -6552.869} C_VEL
LIN {X 0,Y 491.656,Z 535.301,A -85,B 0,C 180,E1 -6553.387,E2 -6553.387} C_VEL
LIN {X 0,Y 491.158,Z 547.667,A -85,B 0,C 180,E1 -6554.015,E2 -6554.015} C_VEL
LIN {X 0,Y 490.587,Z 560.506,A -85,B 0,C 180,E1 -6554.844,E2 -6554.844} C_VEL
LIN {X 0,Y 490.012,Z 572.242,A -85,B 0,C 180,E1 -6555.781,E2 -6555.781} C_VEL
LIN {X 0,Y 489.466,Z 583.97,A -85,B 0,C 180,E1 -6556.929,E2 -6556.929} C_VEL
LIN {X 0,Y 489.106,Z 593.492,A -85,B 0,C 180,E1 -6558.06,E2 -6558.06} C_VEL
LIN {X 0,Y 488.661,Z 603.118,A -85,B 0,C 180,E1 -6559.433,E2 -6559.433} C_VEL
LIN {X 0,Y 488.332,Z 611.413,A -85,B 0,C 180,E1 -6560.89,E2 -6560.89} C_VEL
LIN {X 0,Y 488.147,Z 617.214,A -85,B 0,C 180,E1 -6562.138,E2 -6562.138} C_VEL
LIN {X 0,Y 488.005,Z 622.612,A -85,B 0,C 180,E1 -6563.568,E2 -6563.568} C_VEL
LIN {X 0,Y 487.961,Z 626.903,A -85,B 0,C 180,E1 -6565.042,E2 -6565.042} C_VEL
LIN {X 0,Y 487.956,Z 630.331,A -85,B 0,C 180,E1 -6566.697,E2 -6566.697} C_VEL
LIN {X 0,Y 487.888,Z 632.355,A -85,B 0,C 180,E1 -6568.348,E2 -6568.348} C_VEL
LIN {X 0,Y 487.817,Z 633.022,A -85,B 0,C 180,E1 -6569.999,E2 -6569.999} C_VEL
LIN {X 0,Y 487.888,Z 632.348,A -85,B 0,C 180,E1 -6571.65,E2 -6571.65} C_VEL
LIN {X 0,Y 487.955,Z 630.317,A -85,B 0,C 180,E1 -6573.302,E2 -6573.302} C_VEL
LIN {X 0,Y 487.96,Z 626.878,A -85,B 0,C 180,E1 -6574.957,E2 -6574.957} C_VEL
LIN {X 0,Y 488.04,Z 621.934,A -85,B 0,C 180,E1 -6576.615,E2 -6576.615} C_VEL
LIN {X 0,Y 488.223,Z 615.339,A -85,B 0,C 180,E1 -6578.276,E2 -6578.276} C_VEL
LIN {X 0,Y 488.438,Z 608.002,A -85,B 0,C 180,E1 -6579.733,E2 -6579.733} C_VEL
LIN {X 0,Y 488.859,Z 598.92,A -85,B 0,C 180,E1 -6581.19,E2 -6581.19} C_VEL
LIN {X 0,Y 489.261,Z 589.393,A -85,B 0,C 180,E1 -6582.442,E2 -6582.442} C_VEL
LIN {X 0,Y 489.682,Z 578.86,A -85,B 0,C 180,E1 -6583.592,E2 -6583.592} C_VEL
LIN {X 0,Y 490.26,Z 567.248,A -85,B 0,C 180,E1 -6584.634,E2 -6584.634} C_VEL
LIN {X 0,Y 490.875,Z 554.374,A -85,B 0,C 180,E1 -6585.571,E2 -6585.571} C_VEL
LIN {X 0,Y 491.392,Z 541.862,A -85,B 0,C 180,E1 -6586.297,E2 -6586.297} C_VEL
LIN {X 0,Y 491.873,Z 528.595,A -85,B 0,C 180,E1 -6586.892,E2 -6586.892} C_VEL
LIN {X 0,Y 492.293,Z 515.293,A -85,B 0,C 180,E1 -6587.327,E2 -6587.327} C_VEL
LIN {X 0,Y 492.547,Z 501.448,A -85,B 0,C 180,E1 -6587.623,E2 -6587.623} C_VEL
LIN {X 0,Y 493.397,Z 387.169,A -85,B 0,C 180,E1 -6589.322,E2 -6589.322} C_VEL
LIN {X 0,Y 490.275,Z 368.876,A -85,B 0,C 180,E1 -6589.739,E2 -6589.739} C_VEL
LIN {X 0,Y 491.057,Z 348.902,A -85,B 0,C 180,E1 -6592.731,E2 -6592.731} C_VEL
LIN {X 0,Y 491.751,Z 332.962,A -85,B 0,C 180,E1 -6595.161,E2 -6595.161} C_VEL
LIN {X 0,Y 489.73,Z 322.441,A -85,B 0,C 180,E1 -6596.933,E2 -6596.933} C_VEL
LIN {X 0,Y 488.764,Z 318.229,A -85,B 0,C 180,E1 -6597.685,E2 -6597.685} C_VEL
LIN {X 0,Y 488.708,Z 318.234,A -85,B 0,C 180,E1 -6600.362,E2 -6600.362} C_VEL
LIN {X 0,Y 488.733,Z 318.228,A -85,B 0,C 180,E1 -6603.483,E2 -6603.483} C_VEL
LIN {X 0,Y 488.686,Z 318.234,A -85,B 0,C 180,E1 -6606.355,E2 -6606.355} C_VEL
LIN {X 0,Y 488.734,Z 318.231,A -85,B 0,C 180,E1 -6609.25,E2 -6609.25} C_VEL
LIN {X 0,Y 488.708,Z 318.228,A -85,B 0,C 180,E1 -6611.6,E2 -6611.6} C_VEL
LIN {X 0,Y 488.708,Z 318.232,A -85,B 0,C 180,E1 -6614.8,E2 -6614.8} C_VEL
LIN {X 0,Y 488.69,Z 318.233,A -85,B 0,C 180,E1 -6617.474,E2 -6617.474} C_VEL
LIN {X 0,Y 488.727,Z 318.225,A -85,B 0,C 180,E1 -6619.676,E2 -6619.676} C_VEL
LIN {X 0,Y 488.677,Z 318.238,A -85,B 0,C 180,E1 -6622.841,E2 -6622.841} C_VEL
LIN {X 0,Y 488.728,Z 318.23,A -85,B 0,C 180,E1 -6625.887,E2 -6625.887} C_VEL
LIN {X 0,Y 488.689,Z 318.235,A -85,B 0,C 180,E1 -6628.82,E2 -6628.82} C_VEL
LIN {X 0,Y 488.741,Z 318.227,A -85,B 0,C 180,E1 -6631.671,E2 -6631.671} C_VEL
LIN {X 0,Y 488.735,Z 318.233,A -85,B 0,C 180,E1 -6634.443,E2 -6634.443} C_VEL
LIN {X 0,Y 488.714,Z 318.226,A -85,B 0,C 180,E1 -6637.152,E2 -6637.152} C_VEL
LIN {X 0,Y 488.717,Z 318.233,A -85,B 0,C 180,E1 -6639.81,E2 -6639.81} C_VEL
LIN {X 0,Y 488.726,Z 318.232,A -85,B 0,C 180,E1 -6642.423,E2 -6642.423} C_VEL
LIN {X 0,Y 488.753,Z 318.221,A -85,B 0,C 180,E1 -6644.999,E2 -6644.999} C_VEL
LIN {X 0,Y 488.796,Z 318.218,A -85,B 0,C 180,E1 -6648.387,E2 -6648.387} C_VEL
LIN {X 0,Y 488.806,Z 318.225,A -85,B 0,C 180,E1 -6651.733,E2 -6651.733} C_VEL
LIN {X 0,Y 488.834,Z 318.218,A -85,B 0,C 180,E1 -6654.224,E2 -6654.224} C_VEL
LIN {X 0,Y 488.939,Z 318.203,A -85,B 0,C 180,E1 -6657.528,E2 -6657.528} C_VEL
LIN {X 0,Y 488.93,Z 318.205,A -85,B 0,C 180,E1 -6660,E2 -6660} C_VEL
LIN {X 0,Y 488.939,Z 318.202,A -85,B 0,C 180,E1 -6662.471,E2 -6662.471} C_VEL
LIN {X 0,Y 488.794,Z 318.225,A -85,B 0,C 180,E1 -6665.776,E2 -6665.776} C_VEL
LIN {X 0,Y 488.748,Z 318.224,A -85,B 0,C 180,E1 -6668.267,E2 -6668.267} C_VEL
LIN {X 0,Y 488.793,Z 318.224,A -85,B 0,C 180,E1 -6671.612,E2 -6671.612} C_VEL
LIN {X 0,Y 488.764,Z 318.227,A -85,B 0,C 180,E1 -6675.554,E2 -6675.554} C_VEL
LIN {X 0,Y 488.733,Z 318.227,A -85,B 0,C 180,E1 -6678.443,E2 -6678.443} C_VEL
LIN {X 0,Y 488.696,Z 318.238,A -85,B 0,C 180,E1 -6681.071,E2 -6681.071} C_VEL
LIN {X 0,Y 488.658,Z 318.239,A -85,B 0,C 180,E1 -6683.747,E2 -6683.747} C_VEL
LIN {X 0,Y 488.713,Z 318.237,A -85,B 0,C 180,E1 -6686.928,E2 -6686.928} C_VEL
LIN {X 0,Y 488.694,Z 318.235,A -85,B 0,C 180,E1 -6690.362,E2 -6690.362} C_VEL
LIN {X 0,Y 488.719,Z 318.234,A -85,B 0,C 180,E1 -6693.483,E2 -6693.483} C_VEL
LIN {X 0,Y 488.672,Z 318.238,A -85,B 0,C 180,E1 -6696.355,E2 -6696.355} C_VEL
LIN {X 0,Y 488.691,Z 318.234,A -85,B 0,C 180,E1 -6699.255,E2 -6699.255} C_VEL
LIN {X 0,Y 488.697,Z 318.231,A -85,B 0,C 180,E1 -6701.6,E2 -6701.6} C_VEL
LIN {X 0,Y 488.692,Z 318.24,A -85,B 0,C 180,E1 -6704.803,E2 -6704.803} C_VEL
LIN {X 0,Y 488.683,Z 318.239,A -85,B 0,C 180,E1 -6707.475,E2 -6707.475} C_VEL
LIN {X 0,Y 488.739,Z 318.326,A -85,B 0,C 180,E1 -6708.974,E2 -6708.974} C_VEL
LIN {X 0,Y 490.595,Z 328.019,A -85,B 0,C 180,E1 -6710.928,E2 -6710.928} C_VEL
LIN {X 0,Y 490.391,Z 335.464,A -85,B 0,C 180,E1 -6712.317,E2 -6712.317} C_VEL
LIN {X 0,Y 493.609,Z 349.843,A -85,B 0,C 180,E1 -6712.693,E2 -6712.693} C_VEL
LIN {X 0,Y 493.064,Z 419.707,A -85,B 0,C 180,E1 -6713.735,E2 -6713.735} C_VEL
LIN {X 0,Y 492.343,Z 425.553,A -85,B 0,C 180,E1 -6713.795,E2 -6713.795} C_VEL
LIN {X 0,Y 486.768,Z 444.577,A -85,B 0,C 180,E1 -6713.861,E2 -6713.861} C_VEL
LIN {X 0,Y 486.09,Z 450.42,A -85,B 0,C 180,E1 -6713.924,E2 -6713.924} C_VEL
LIN {X 0,Y 485.821,Z 474.034,A -85,B 0,C 180,E1 -6714.316,E2 -6714.316} C_VEL
LIN {X 0,Y 485.466,Z 488.861,A -85,B 0,C 180,E1 -6714.743,E2 -6714.743} C_VEL
LIN {X 0,Y 485.118,Z 501.853,A -85,B 0,C 180,E1 -6715.284,E2 -6715.284} C_VEL
LIN {X 0,Y 484.582,Z 514.187,A -85,B 0,C 180,E1 -6715.95,E2 -6715.95} C_VEL
LIN {X 0,Y 484.018,Z 526.158,A -85,B 0,C 180,E1 -6716.762,E2 -6716.762} C_VEL
LIN {X 0,Y 483.435,Z 537.492,A -85,B 0,C 180,E1 -6717.708,E2 -6717.708} C_VEL
LIN {X 0,Y 482.884,Z 548.834,A -85,B 0,C 180,E1 -6718.862,E2 -6718.862} C_VEL
LIN {X 0,Y 482.367,Z 558.581,A -85,B 0,C 180,E1 -6720.066,E2 -6720.066} C_VEL
LIN {X 0,Y 481.865,Z 567.915,A -85,B 0,C 180,E1 -6721.469,E2 -6721.469} C_VEL
LIN {X 0,Y 481.487,Z 575.763,A -85,B 0,C 180,E1 -6722.92,E2 -6722.92} C_VEL
LIN {X 0,Y 481.177,Z 582.517,A -85,B 0,C 180,E1 -6724.479,E2 -6724.479} C_VEL
LIN {X 0,Y 481.028,Z 587.248,A -85,B 0,C 180,E1 -6725.853,E2 -6725.853} C_VEL
LIN {X 0,Y 480.901,Z 590.441,A -85,B 0,C 180,E1 -6727.027,E2 -6727.027} C_VEL
LIN {X 0,Y 480.795,Z 593.548,A -85,B 0,C 180,E1 -6728.567,E2 -6728.567} C_VEL
LIN {X 0,Y 480.787,Z 594.828,A -85,B 0,C 180,E1 -6729.463,E2 -6729.463} C_VEL
LIN {X 0,Y 480.741,Z 596.243,A -85,B 0,C 180,E1 -6731.24,E2 -6731.24} C_VEL
LIN {X 0,Y 480.775,Z 596.381,A -85,B 0,C 180,E1 -6732.124,E2 -6732.124} C_VEL
LIN {X 0,Y 480.694,Z 595.582,A -85,B 0,C 180,E1 -6733.873,E2 -6733.873} C_VEL
LIN {X 0,Y 480.832,Z 593.356,A -85,B 0,C 180,E1 -6735.613,E2 -6735.613} C_VEL
LIN {X 0,Y 480.933,Z 589.696,A -85,B 0,C 180,E1 -6737.339,E2 -6737.339} C_VEL
LIN {X 0,Y 481.075,Z 585.948,A -85,B 0,C 180,E1 -6738.626,E2 -6738.626} C_VEL
LIN {X 0,Y 481.21,Z 581.305,A -85,B 0,C 180,E1 -6739.907,E2 -6739.907} C_VEL
LIN {X 0,Y 481.514,Z 574.547,A -85,B 0,C 180,E1 -6741.397,E2 -6741.397} C_VEL
LIN {X 0,Y 481.899,Z 566.161,A -85,B 0,C 180,E1 -6742.882,E2 -6742.882} C_VEL
LIN {X 0,Y 482.348,Z 557.472,A -85,B 0,C 180,E1 -6744.147,E2 -6744.147} C_VEL
LIN {X 0,Y 482.906,Z 546.958,A -85,B 0,C 180,E1 -6745.41,E2 -6745.41} C_VEL
LIN {X 0,Y 483.428,Z 536.389,A -85,B 0,C 180,E1 -6746.458,E2 -6746.458} C_VEL
LIN {X 0,Y 484.043,Z 524.844,A -85,B 0,C 180,E1 -6747.4,E2 -6747.4} C_VEL
LIN {X 0,Y 484.603,Z 512.207,A -85,B 0,C 180,E1 -6748.235,E2 -6748.235} C_VEL
LIN {X 0,Y 485.17,Z 498.535,A -85,B 0,C 180,E1 -6748.937,E2 -6748.937} C_VEL
LIN {X 0,Y 485.55,Z 484.547,A -85,B 0,C 180,E1 -6749.469,E2 -6749.469} C_VEL
LIN {X 0,Y 485.836,Z 470.557,A -85,B 0,C 180,E1 -6749.824,E2 -6749.824} C_VEL
LIN {X 0,Y 486.81,Z 350.884,A -85,B 0,C 180,E1 -6751.639,E2 -6751.639} C_VEL
LIN {X 0,Y 483.455,Z 335.442,A -85,B 0,C 180,E1 -6752.037,E2 -6752.037} C_VEL
LIN {X 0,Y 483.563,Z 328.544,A -85,B 0,C 180,E1 -6753.333,E2 -6753.333} C_VEL
LIN {X 0,Y 481.778,Z 319.101,A -85,B 0,C 180,E1 -6755.232,E2 -6755.232} C_VEL
LIN {X 0,Y 481.775,Z 319.102,A -85,B 0,C 180,E1 -6757.545,E2 -6757.545} C_VEL
LIN {X 0,Y 481.703,Z 319.107,A -85,B 0,C 180,E1 -6760.084,E2 -6760.084} C_VEL
LIN {X 0,Y 481.68,Z 319.106,A -85,B 0,C 180,E1 -6762.643,E2 -6762.643} C_VEL
LIN {X 0,Y 481.723,Z 319.103,A -85,B 0,C 180,E1 -6765.659,E2 -6765.659} C_VEL
LIN {X 0,Y 481.706,Z 319.104,A -85,B 0,C 180,E1 -6768.723,E2 -6768.723} C_VEL
LIN {X 0,Y 481.643,Z 319.115,A -85,B 0,C 180,E1 -6771.395,E2 -6771.395} C_VEL
LIN {X 0,Y 481.645,Z 319.109,A -85,B 0,C 180,E1 -6774.115,E2 -6774.115} C_VEL
LIN {X 0,Y 481.65,Z 319.116,A -85,B 0,C 180,E1 -6777.117,E2 -6777.117} C_VEL
LIN {X 0,Y 481.65,Z 319.109,A -85,B 0,C 180,E1 -6779.744,E2 -6779.744} C_VEL
LIN {X 0,Y 481.632,Z 319.116,A -85,B 0,C 180,E1 -6782.678,E2 -6782.678} C_VEL
LIN {X 0,Y 481.646,Z 319.114,A -85,B 0,C 180,E1 -6785.202,E2 -6785.202} C_VEL
LIN {X 0,Y 481.625,Z 319.112,A -85,B 0,C 180,E1 -6788.003,E2 -6788.003} C_VEL
LIN {X 0,Y 481.621,Z 319.117,A -85,B 0,C 180,E1 -6791.046,E2 -6791.046} C_VEL
LIN {X 0,Y 481.649,Z 319.113,A -85,B 0,C 180,E1 -6794.459,E2 -6794.459} C_VEL
LIN {X 0,Y 481.61,Z 319.12,A -85,B 0,C 180,E1 -6796.856,E2 -6796.856} C_VEL
LIN {X 0,Y 481.628,Z 319.113,A -85,B 0,C 180,E1 -6800.055,E2 -6800.055} C_VEL
LIN {X 0,Y 481.603,Z 319.116,A -85,B 0,C 180,E1 -6803.252,E2 -6803.252} C_VEL
LIN {X 0,Y 481.671,Z 319.111,A -85,B 0,C 180,E1 -6806.327,E2 -6806.327} C_VEL
LIN {X 0,Y 481.633,Z 319.111,A -85,B 0,C 180,E1 -6809.422,E2 -6809.422} C_VEL
LIN {X 0,Y 481.647,Z 319.114,A -85,B 0,C 180,E1 -6812.165,E2 -6812.165} C_VEL
LIN {X 0,Y 481.673,Z 319.108,A -85,B 0,C 180,E1 -6814.968,E2 -6814.968} C_VEL
LIN {X 0,Y 481.637,Z 319.111,A -85,B 0,C 180,E1 -6817.705,E2 -6817.705} C_VEL
LIN {X 0,Y 481.696,Z 319.111,A -85,B 0,C 180,E1 -6820.393,E2 -6820.393} C_VEL
LIN {X 0,Y 481.618,Z 319.113,A -85,B 0,C 180,E1 -6823.032,E2 -6823.032} C_VEL
LIN {X 0,Y 481.676,Z 319.107,A -85,B 0,C 180,E1 -6825.639,E2 -6825.639} C_VEL
LIN {X 0,Y 481.753,Z 319.104,A -85,B 0,C 180,E1 -6828.215,E2 -6828.215} C_VEL
LIN {X 0,Y 481.738,Z 319.1,A -85,B 0,C 180,E1 -6831.612,E2 -6831.612} C_VEL
LIN {X 0,Y 481.795,Z 319.099,A -85,B 0,C 180,E1 -6834.14,E2 -6834.14} C_VEL
LIN {X 0,Y 481.921,Z 319.077,A -85,B 0,C 180,E1 -6837.493,E2 -6837.493} C_VEL
LIN {X 0,Y 481.941,Z 319.081,A -85,B 0,C 180,E1 -6840,E2 -6840} C_VEL
LIN {X 0,Y 481.92,Z 319.077,A -85,B 0,C 180,E1 -6842.508,E2 -6842.508} C_VEL
LIN {X 0,Y 481.8,Z 319.098,A -85,B 0,C 180,E1 -6845.861,E2 -6845.861} C_VEL
LIN {X 0,Y 481.764,Z 319.096,A -85,B 0,C 180,E1 -6848.389,E2 -6848.389} C_VEL
LIN {X 0,Y 481.754,Z 319.104,A -85,B 0,C 180,E1 -6851.785,E2 -6851.785} C_VEL
LIN {X 0,Y 481.746,Z 319.099,A -85,B 0,C 180,E1 -6855.224,E2 -6855.224} C_VEL
LIN {X 0,Y 481.716,Z 319.101,A -85,B 0,C 180,E1 -6858.722,E2 -6858.722} C_VEL
LIN {X 0,Y 481.65,Z 319.114,A -85,B 0,C 180,E1 -6861.395,E2 -6861.395} C_VEL
LIN {X 0,Y 481.664,Z 319.109,A -85,B 0,C 180,E1 -6864.114,E2 -6864.114} C_VEL
LIN {X 0,Y 481.75,Z 319.099,A -85,B 0,C 180,E1 -6867.139,E2 -6867.139} C_VEL
LIN {X 0,Y 481.682,Z 319.11,A -85,B 0,C 180,E1 -6869.741,E2 -6869.741} C_VEL
LIN {X 0,Y 481.676,Z 319.106,A -85,B 0,C 180,E1 -6872.674,E2 -6872.674} C_VEL
LIN {X 0,Y 481.664,Z 319.113,A -85,B 0,C 180,E1 -6875.204,E2 -6875.204} C_VEL
LIN {X 0,Y 481.673,Z 319.108,A -85,B 0,C 180,E1 -6878.859,E2 -6878.859} C_VEL
LIN {X 0,Y 481.656,Z 319.109,A -85,B 0,C 180,E1 -6881.913,E2 -6881.913} C_VEL
LIN {X 0,Y 481.664,Z 319.107,A -85,B 0,C 180,E1 -6884.457,E2 -6884.457} C_VEL
LIN {X 0,Y 481.651,Z 319.11,A -85,B 0,C 180,E1 -6887.839,E2 -6887.839} C_VEL
LIN {X 0,Y 481.685,Z 319.107,A -85,B 0,C 180,E1 -6890.651,E2 -6890.651} C_VEL
LIN {X 0,Y 481.631,Z 319.116,A -85,B 0,C 180,E1 -6893.376,E2 -6893.376} C_VEL
LIN {X 0,Y 481.714,Z 319.101,A -85,B 0,C 180,E1 -6896.33,E2 -6896.33} C_VEL
LIN {X 0,Y 481.653,Z 319.118,A -85,B 0,C 180,E1 -6899.417,E2 -6899.417} C_VEL
LIN {X 0,Y 481.746,Z 319.282,A -85,B 0,C 180,E1 -6902.215,E2 -6902.215} C_VEL
LIN {X 0,Y 484.608,Z 332.415,A -85,B 0,C 180,E1 -6904.44,E2 -6904.44} C_VEL
LIN {X 0,Y 484.658,Z 338.292,A -85,B 0,C 180,E1 -6905.36,E2 -6905.36} C_VEL
LIN {X 0,Y 483.768,Z 359.056,A -85,B 0,C 180,E1 -6908.523,E2 -6908.523} C_VEL
LIN {X 0,Y 483.358,Z 368.877,A -85,B 0,C 180,E1 -6910.001,E2 -6910.001} C_VEL
LIN {X 0,Y 486.728,Z 389.336,A -85,B 0,C 180,E1 -6910.456,E2 -6910.456} C_VEL
LIN {X 0,Y 485.662,Z 507.69,A -85,B 0,C 180,E1 -6912.254,E2 -6912.254} C_VEL
LIN {X 0,Y 485.219,Z 522.298,A -85,B 0,C 180,E1 -6912.65,E2 -6912.65} C_VEL
LIN {X 0,Y 484.791,Z 536.352,A -85,B 0,C 180,E1 -6913.214,E2 -6913.214} C_VEL
LIN {X 0,Y 484.229,Z 549.146,A -85,B 0,C 180,E1 -6913.892,E2 -6913.892} C_VEL
LIN {X 0,Y 483.61,Z 561.596,A -85,B 0,C 180,E1 -6914.728,E2 -6914.728} C_VEL
LIN {X 0,Y 482.942,Z 574.275,A -85,B 0,C 180,E1 -6915.784,E2 -6915.784} C_VEL
LIN {X 0,Y 482.428,Z 585.583,A -85,B 0,C 180,E1 -6916.949,E2 -6916.949} C_VEL
LIN {X 0,Y 481.945,Z 595.707,A -85,B 0,C 180,E1 -6918.219,E2 -6918.219} C_VEL
LIN {X 0,Y 481.562,Z 604.117,A -85,B 0,C 180,E1 -6919.488,E2 -6919.488} C_VEL
LIN {X 0,Y 481.253,Z 612.157,A -85,B 0,C 180,E1 -6920.967,E2 -6920.967} C_VEL
LIN {X 0,Y 481.007,Z 618.628,A -85,B 0,C 180,E1 -6922.443,E2 -6922.443} C_VEL
LIN {X 0,Y 480.9,Z 624.366,A -85,B 0,C 180,E1 -6924.128,E2 -6924.128} C_VEL
LIN {X 0,Y 480.815,Z 628.527,A -85,B 0,C 180,E1 -6925.808,E2 -6925.808} C_VEL
LIN {X 0,Y 480.879,Z 630.064,A -85,B 0,C 180,E1 -6926.648,E2 -6926.648} C_VEL
LIN {X 0,Y 480.818,Z 632.088,A -85,B 0,C 180,E1 -6928.324,E2 -6928.324} C_VEL
LIN {X 0,Y 480.741,Z 632.754,A -85,B 0,C 180,E1 -6929.999,E2 -6929.999} C_VEL
LIN {X 0,Y 480.818,Z 632.079,A -85,B 0,C 180,E1 -6931.674,E2 -6931.674} C_VEL
LIN {X 0,Y 480.879,Z 630.046,A -85,B 0,C 180,E1 -6933.351,E2 -6933.351} C_VEL
LIN {X 0,Y 480.891,Z 626.605,A -85,B 0,C 180,E1 -6935.03,E2 -6935.03} C_VEL
LIN {X 0,Y 480.959,Z 621.656,A -85,B 0,C 180,E1 -6936.712,E2 -6936.712} C_VEL
LIN {X 0,Y 481.139,Z 615.061,A -85,B 0,C 180,E1 -6938.398,E2 -6938.398} C_VEL
LIN {X 0,Y 481.372,Z 607.727,A -85,B 0,C 180,E1 -6939.877,E2 -6939.877} C_VEL
LIN {X 0,Y 481.838,Z 598.653,A -85,B 0,C 180,E1 -6941.355,E2 -6941.355} C_VEL
LIN {X 0,Y 482.261,Z 589.135,A -85,B 0,C 180,E1 -6942.626,E2 -6942.626} C_VEL
LIN {X 0,Y 482.739,Z 578.605,A -85,B 0,C 180,E1 -6943.791,E2 -6943.791} C_VEL
LIN {X 0,Y 483.37,Z 566.998,A -85,B 0,C 180,E1 -6944.847,E2 -6944.847} C_VEL
LIN {X 0,Y 484.013,Z 554.128,A -85,B 0,C 180,E1 -6945.798,E2 -6945.798} C_VEL
LIN {X 0,Y 484.527,Z 542.285,A -85,B 0,C 180,E1 -6946.498,E2 -6946.498} C_VEL
LIN {X 0,Y 485.036,Z 528.371,A -85,B 0,C 180,E1 -6947.138,E2 -6947.138} C_VEL
LIN {X 0,Y 485.556,Z 514.09,A -85,B 0,C 180,E1 -6947.605,E2 -6947.605} C_VEL
LIN {X 0,Y 485.805,Z 499.786,A -85,B 0,C 180,E1 -6947.903,E2 -6947.903} C_VEL
LIN {X 0,Y 486.741,Z 388.2,A -85,B 0,C 180,E1 -6949.586,E2 -6949.586} C_VEL
LIN {X 0,Y 483.381,Z 368.543,A -85,B 0,C 180,E1 -6950.051,E2 -6950.051} C_VEL
LIN {X 0,Y 484.147,Z 350.177,A -85,B 0,C 180,E1 -6952.848,E2 -6952.848} C_VEL
LIN {X 0,Y 484.881,Z 334.287,A -85,B 0,C 180,E1 -6955.313,E2 -6955.313} C_VEL
LIN {X 0,Y 482.775,Z 323.635,A -85,B 0,C 180,E1 -6957.143,E2 -6957.143} C_VEL
LIN {X 0,Y 481.708,Z 319.108,A -85,B 0,C 180,E1 -6957.978,E2 -6957.978} C_VEL
LIN {X 0,Y 481.644,Z 319.116,A -85,B 0,C 180,E1 -6960.71,E2 -6960.71} C_VEL
LIN {X 0,Y 481.694,Z 319.104,A -85,B 0,C 180,E1 -6963.732,E2 -6963.732} C_VEL
LIN {X 0,Y 481.626,Z 319.116,A -85,B 0,C 180,E1 -6966.746,E2 -6966.746} C_VEL
LIN {X 0,Y 481.684,Z 319.107,A -85,B 0,C 180,E1 -6969.938,E2 -6969.938} C_VEL
LIN {X 0,Y 481.635,Z 319.115,A -85,B 0,C 180,E1 -6973.299,E2 -6973.299} C_VEL
LIN {X 0,Y 481.654,Z 319.104,A -85,B 0,C 180,E1 -6975.64,E2 -6975.64} C_VEL
LIN {X 0,Y 481.658,Z 319.109,A -85,B 0,C 180,E1 -6978.958,E2 -6978.958} C_VEL
LIN {X 0,Y 481.65,Z 319.109,A -85,B 0,C 180,E1 -6981.992,E2 -6981.992} C_VEL
LIN {X 0,Y 481.686,Z 319.106,A -85,B 0,C 180,E1 -6985.317,E2 -6985.317} C_VEL
LIN {X 0,Y 481.641,Z 319.116,A -85,B 0,C 180,E1 -6988.311,E2 -6988.311} C_VEL
LIN {X 0,Y 481.7,Z 319.103,A -85,B 0,C 180,E1 -6991.218,E2 -6991.218} C_VEL
LIN {X 0,Y 481.695,Z 319.106,A -85,B 0,C 180,E1 -6994.042,E2 -6994.042} C_VEL
LIN {X 0,Y 481.666,Z 319.105,A -85,B 0,C 180,E1 -6996.811,E2 -6996.811} C_VEL
LIN {X 0,Y 481.688,Z 319.106,A -85,B 0,C 180,E1 -6999.502,E2 -6999.502} C_VEL
LIN {X 0,Y 481.699,Z 319.11,A -85,B 0,C 180,E1 -7002.158,E2 -7002.158} C_VEL
LIN {X 0,Y 481.734,Z 319.096,A -85,B 0,C 180,E1 -7004.775,E2 -7004.775} C_VEL
LIN {X 0,Y 481.742,Z 319.099,A -85,B 0,C 180,E1 -7008.215,E2 -7008.215} C_VEL
LIN {X 0,Y 481.752,Z 319.102,A -85,B 0,C 180,E1 -7011.611,E2 -7011.611} C_VEL
LIN {X 0,Y 481.795,Z 319.096,A -85,B 0,C 180,E1 -7014.139,E2 -7014.139} C_VEL
LIN {X 0,Y 481.905,Z 319.079,A -85,B 0,C 180,E1 -7017.492,E2 -7017.492} C_VEL
LIN {X 0,Y 481.9,Z 319.081,A -85,B 0,C 180,E1 -7020,E2 -7020} C_VEL
LIN {X 0,Y 481.905,Z 319.078,A -85,B 0,C 180,E1 -7022.507,E2 -7022.507} C_VEL
LIN {X 0,Y 481.755,Z 319.101,A -85,B 0,C 180,E1 -7025.861,E2 -7025.861} C_VEL
LIN {X 0,Y 481.707,Z 319.101,A -85,B 0,C 180,E1 -7028.389,E2 -7028.389} C_VEL
LIN {X 0,Y 481.739,Z 319.1,A -85,B 0,C 180,E1 -7031.785,E2 -7031.785} C_VEL
LIN {X 0,Y 481.725,Z 319.107,A -85,B 0,C 180,E1 -7035.224,E2 -7035.224} C_VEL
LIN {X 0,Y 481.694,Z 319.106,A -85,B 0,C 180,E1 -7038.722,E2 -7038.722} C_VEL
LIN {X 0,Y 481.634,Z 319.116,A -85,B 0,C 180,E1 -7041.395,E2 -7041.395} C_VEL
LIN {X 0,Y 481.637,Z 319.112,A -85,B 0,C 180,E1 -7044.115,E2 -7044.115} C_VEL
LIN {X 0,Y 481.681,Z 319.111,A -85,B 0,C 180,E1 -7047.126,E2 -7047.126} C_VEL
LIN {X 0,Y 481.656,Z 319.112,A -85,B 0,C 180,E1 -7049.742,E2 -7049.742} C_VEL
LIN {X 0,Y 481.66,Z 319.112,A -85,B 0,C 180,E1 -7052.675,E2 -7052.675} C_VEL
LIN {X 0,Y 481.626,Z 319.115,A -85,B 0,C 180,E1 -7055.71,E2 -7055.71} C_VEL
LIN {X 0,Y 481.661,Z 319.113,A -85,B 0,C 180,E1 -7058.86,E2 -7058.86} C_VEL
LIN {X 0,Y 481.643,Z 319.109,A -85,B 0,C 180,E1 -7061.913,E2 -7061.913} C_VEL
LIN {X 0,Y 481.646,Z 319.114,A -85,B 0,C 180,E1 -7064.458,E2 -7064.458} C_VEL
LIN {X 0,Y 481.639,Z 319.117,A -85,B 0,C 180,E1 -7067.84,E2 -7067.84} C_VEL
LIN {X 0,Y 481.692,Z 319.241,A -85,B 0,C 180,E1 -7068.725,E2 -7068.725} C_VEL
LIN {X 0,Y 483.69,Z 329.336,A -85,B 0,C 180,E1 -7070.8,E2 -7070.8} C_VEL
LIN {X 0,Y 483.524,Z 335.774,A -85,B 0,C 180,E1 -7072.021,E2 -7072.021} C_VEL
LIN {X 0,Y 486.933,Z 350.9,A -85,B 0,C 180,E1 -7072.419,E2 -7072.419} C_VEL
LIN {X 0,Y 486.09,Z 450.42,A -85,B 0,C 180,E1 -7073.924,E2 -7073.924} C_VEL
LIN {X 0,Y 485.37,Z 456.284,A -85,B 0,C 180,E1 -7073.983,E2 -7073.983} C_VEL
LIN {X 0,Y 479.608,Z 475.255,A -85,B 0,C 180,E1 -7074.09,E2 -7074.09} C_VEL
LIN {X 0,Y 479.009,Z 480.995,A -85,B 0,C 180,E1 -7074.221,E2 -7074.221} C_VEL
LIN {X 0,Y 478.583,Z 494.222,A -85,B 0,C 180,E1 -7074.676,E2 -7074.676} C_VEL
LIN {X 0,Y 478.079,Z 508.412,A -85,B 0,C 180,E1 -7075.352,E2 -7075.352} C_VEL
LIN {X 0,Y 477.523,Z 520.845,A -85,B 0,C 180,E1 -7076.123,E2 -7076.123} C_VEL
LIN {X 0,Y 476.803,Z 533.626,A -85,B 0,C 180,E1 -7077.113,E2 -7077.113} C_VEL
LIN {X 0,Y 476.217,Z 544.541,A -85,B 0,C 180,E1 -7078.158,E2 -7078.158} C_VEL
LIN {X 0,Y 475.633,Z 554.85,A -85,B 0,C 180,E1 -7079.352,E2 -7079.352} C_VEL
LIN {X 0,Y 475.031,Z 565.023,A -85,B 0,C 180,E1 -7080.796,E2 -7080.796} C_VEL
LIN {X 0,Y 474.579,Z 573.098,A -85,B 0,C 180,E1 -7082.195,E2 -7082.195} C_VEL
LIN {X 0,Y 474.25,Z 579.753,A -85,B 0,C 180,E1 -7083.605,E2 -7083.605} C_VEL
LIN {X 0,Y 474.047,Z 585.41,A -85,B 0,C 180,E1 -7085.097,E2 -7085.097} C_VEL
LIN {X 0,Y 473.91,Z 589.348,A -85,B 0,C 180,E1 -7086.398,E2 -7086.398} C_VEL
LIN {X 0,Y 473.793,Z 591.557,A -85,B 0,C 180,E1 -7087.316,E2 -7087.316} C_VEL
LIN {X 0,Y 473.71,Z 594.736,A -85,B 0,C 180,E1 -7089.142,E2 -7089.142} C_VEL
LIN {X 0,Y 473.642,Z 596.367,A -85,B 0,C 180,E1 -7090.948,E2 -7090.948} C_VEL
LIN {X 0,Y 473.688,Z 596.629,A -85,B 0,C 180,E1 -7091.847,E2 -7091.847} C_VEL
LIN {X 0,Y 473.608,Z 596.08,A -85,B 0,C 180,E1 -7093.625,E2 -7093.625} C_VEL
LIN {X 0,Y 473.72,Z 594.08,A -85,B 0,C 180,E1 -7095.393,E2 -7095.393} C_VEL
LIN {X 0,Y 473.845,Z 590.623,A -85,B 0,C 180,E1 -7097.146,E2 -7097.146} C_VEL
LIN {X 0,Y 474.001,Z 586.875,A -85,B 0,C 180,E1 -7098.519,E2 -7098.519} C_VEL
LIN {X 0,Y 474.205,Z 580.866,A -85,B 0,C 180,E1 -7100.188,E2 -7100.188} C_VEL
LIN {X 0,Y 474.529,Z 573.944,A -85,B 0,C 180,E1 -7101.698,E2 -7101.698} C_VEL
LIN {X 0,Y 474.942,Z 565.397,A -85,B 0,C 180,E1 -7103.202,E2 -7103.202} C_VEL
LIN {X 0,Y 475.451,Z 556.48,A -85,B 0,C 180,E1 -7104.487,E2 -7104.487} C_VEL
LIN {X 0,Y 476.061,Z 545.718,A -85,B 0,C 180,E1 -7105.768,E2 -7105.768} C_VEL
LIN {X 0,Y 476.641,Z 534.832,A -85,B 0,C 180,E1 -7106.831,E2 -7106.831} C_VEL
LIN {X 0,Y 477.258,Z 522.901,A -85,B 0,C 180,E1 -7107.785,E2 -7107.785} C_VEL
LIN {X 0,Y 477.893,Z 510.451,A -85,B 0,C 180,E1 -7108.583,E2 -7108.583} C_VEL
LIN {X 0,Y 478.407,Z 497.969,A -85,B 0,C 180,E1 -7109.212,E2 -7109.212} C_VEL
LIN {X 0,Y 478.74,Z 484.27,A -85,B 0,C 180,E1 -7109.73,E2 -7109.73} C_VEL
LIN {X 0,Y 479.083,Z 470.356,A -85,B 0,C 180,E1 -7110.08,E2 -7110.08} C_VEL
LIN {X 0,Y 480.118,Z 351.992,A -85,B 0,C 180,E1 -7111.897,E2 -7111.897} C_VEL
LIN {X 0,Y 476.58,Z 335.807,A -85,B 0,C 180,E1 -7112.304,E2 -7112.304} C_VEL
LIN {X 0,Y 476.676,Z 330.135,A -85,B 0,C 180,E1 -7113.382,E2 -7113.382} C_VEL
LIN {X 0,Y 474.777,Z 319.973,A -85,B 0,C 180,E1 -7115.469,E2 -7115.469} C_VEL
LIN {X 0,Y 474.707,Z 319.979,A -85,B 0,C 180,E1 -7118.515,E2 -7118.515} C_VEL
LIN {X 0,Y 474.702,Z 319.975,A -85,B 0,C 180,E1 -7121.963,E2 -7121.963} C_VEL
LIN {X 0,Y 474.678,Z 319.979,A -85,B 0,C 180,E1 -7125.768,E2 -7125.768} C_VEL
LIN {X 0,Y 474.66,Z 319.986,A -85,B 0,C 180,E1 -7129.011,E2 -7129.011} C_VEL
LIN {X 0,Y 474.586,Z 319.99,A -85,B 0,C 180,E1 -7131.73,E2 -7131.73} C_VEL
LIN {X 0,Y 474.623,Z 319.986,A -85,B 0,C 180,E1 -7134.495,E2 -7134.495} C_VEL
LIN {X 0,Y 474.596,Z 319.992,A -85,B 0,C 180,E1 -7137.327,E2 -7137.327} C_VEL
LIN {X 0,Y 474.578,Z 319.99,A -85,B 0,C 180,E1 -7140.233,E2 -7140.233} C_VEL
LIN {X 0,Y 474.606,Z 319.991,A -85,B 0,C 180,E1 -7143.224,E2 -7143.224} C_VEL
LIN {X 0,Y 474.568,Z 319.993,A -85,B 0,C 180,E1 -7146.326,E2 -7146.326} C_VEL
LIN {X 0,Y 474.597,Z 319.988,A -85,B 0,C 180,E1 -7149.644,E2 -7149.644} C_VEL
LIN {X 0,Y 474.574,Z 319.992,A -85,B 0,C 180,E1 -7152.23,E2 -7152.23} C_VEL
LIN {X 0,Y 474.611,Z 319.987,A -85,B 0,C 180,E1 -7155.299,E2 -7155.299} C_VEL
LIN {X 0,Y 474.588,Z 319.991,A -85,B 0,C 180,E1 -7158.212,E2 -7158.212} C_VEL
LIN {X 0,Y 474.582,Z 319.989,A -85,B 0,C 180,E1 -7161.54,E2 -7161.54} C_VEL
LIN {X 0,Y 474.609,Z 319.992,A -85,B 0,C 180,E1 -7164.725,E2 -7164.725} C_VEL
LIN {X 0,Y 474.626,Z 319.984,A -85,B 0,C 180,E1 -7167.787,E2 -7167.787} C_VEL
LIN {X 0,Y 474.591,Z 319.991,A -85,B 0,C 180,E1 -7170.893,E2 -7170.893} C_VEL
LIN {X 0,Y 474.589,Z 319.989,A -85,B 0,C 180,E1 -7173.625,E2 -7173.625} C_VEL
LIN {X 0,Y 474.598,Z 319.992,A -85,B 0,C 180,E1 -7176.653,E2 -7176.653} C_VEL
LIN {X 0,Y 474.645,Z 319.986,A -85,B 0,C 180,E1 -7180.09,E2 -7180.09} C_VEL
LIN {X 0,Y 474.594,Z 319.99,A -85,B 0,C 180,E1 -7182.773,E2 -7182.773} C_VEL
LIN {X 0,Y 474.635,Z 319.983,A -85,B 0,C 180,E1 -7185.421,E2 -7185.421} C_VEL
LIN {X 0,Y 474.707,Z 319.98,A -85,B 0,C 180,E1 -7188.038,E2 -7188.038} C_VEL
LIN {X 0,Y 474.71,Z 319.974,A -85,B 0,C 180,E1 -7191.486,E2 -7191.486} C_VEL
LIN {X 0,Y 474.744,Z 319.969,A -85,B 0,C 180,E1 -7194.904,E2 -7194.904} C_VEL
LIN {X 0,Y 474.887,Z 319.953,A -85,B 0,C 180,E1 -7197.456,E2 -7197.456} C_VEL
LIN {X 0,Y 474.911,Z 319.957,A -85,B 0,C 180,E1 -7200,E2 -7200} C_VEL
LIN {X 0,Y 474.885,Z 319.953,A -85,B 0,C 180,E1 -7202.545,E2 -7202.545} C_VEL
LIN {X 0,Y 474.761,Z 319.975,A -85,B 0,C 180,E1 -7205.948,E2 -7205.948} C_VEL
LIN {X 0,Y 474.729,Z 319.972,A -85,B 0,C 180,E1 -7208.514,E2 -7208.514} C_VEL
LIN {X 0,Y 474.708,Z 319.98,A -85,B 0,C 180,E1 -7211.963,E2 -7211.963} C_VEL
LIN {X 0,Y 474.704,Z 319.979,A -85,B 0,C 180,E1 -7215.456,E2 -7215.456} C_VEL
LIN {X 0,Y 474.669,Z 319.979,A -85,B 0,C 180,E1 -7219.01,E2 -7219.01} C_VEL
LIN {X 0,Y 474.593,Z 319.995,A -85,B 0,C 180,E1 -7221.729,E2 -7221.729} C_VEL
LIN {X 0,Y 474.644,Z 319.982,A -85,B 0,C 180,E1 -7224.494,E2 -7224.494} C_VEL
LIN {X 0,Y 474.685,Z 319.982,A -85,B 0,C 180,E1 -7227.334,E2 -7227.334} C_VEL
LIN {X 0,Y 474.608,Z 319.987,A -85,B 0,C 180,E1 -7230.81,E2 -7230.81} C_VEL
LIN {X 0,Y 474.641,Z 319.984,A -85,B 0,C 180,E1 -7233.984,E2 -7233.984} C_VEL
LIN {X 0,Y 474.57,Z 319.993,A -85,B 0,C 180,E1 -7236.898,E2 -7236.898} C_VEL
LIN {X 0,Y 474.631,Z 319.987,A -85,B 0,C 180,E1 -7239.647,E2 -7239.647} C_VEL
LIN {X 0,Y 474.619,Z 319.988,A -85,B 0,C 180,E1 -7242.934,E2 -7242.934} C_VEL
LIN {X 0,Y 474.613,Z 319.986,A -85,B 0,C 180,E1 -7245.895,E2 -7245.895} C_VEL
LIN {X 0,Y 474.631,Z 319.99,A -85,B 0,C 180,E1 -7249.041,E2 -7249.041} C_VEL
LIN {X 0,Y 474.614,Z 319.987,A -85,B 0,C 180,E1 -7251.704,E2 -7251.704} C_VEL
LIN {X 0,Y 474.629,Z 319.987,A -85,B 0,C 180,E1 -7254.725,E2 -7254.725} C_VEL
LIN {X 0,Y 474.639,Z 319.987,A -85,B 0,C 180,E1 -7257.787,E2 -7257.787} C_VEL
LIN {X 0,Y 474.627,Z 319.995,A -85,B 0,C 180,E1 -7260.884,E2 -7260.884} C_VEL
LIN {X 0,Y 474.712,Z 320.164,A -85,B 0,C 180,E1 -7261.973,E2 -7261.973} C_VEL
LIN {X 0,Y 477.686,Z 333.803,A -85,B 0,C 180,E1 -7264.323,E2 -7264.323} C_VEL
LIN {X 0,Y 477.814,Z 337.934,A -85,B 0,C 180,E1 -7264.983,E2 -7264.983} C_VEL
LIN {X 0,Y 476.888,Z 358.702,A -85,B 0,C 180,E1 -7268.194,E2 -7268.194} C_VEL
LIN {X 0,Y 476.453,Z 368.725,A -85,B 0,C 180,E1 -7269.714,E2 -7269.714} C_VEL
LIN {X 0,Y 480.012,Z 390.291,A -85,B 0,C 180,E1 -7270.198,E2 -7270.198} C_VEL
LIN {X 0,Y 478.884,Z 507.091,A -85,B 0,C 180,E1 -7271.994,E2 -7271.994} C_VEL
LIN {X 0,Y 478.451,Z 521.828,A -85,B 0,C 180,E1 -7272.397,E2 -7272.397} C_VEL
LIN {X 0,Y 477.951,Z 535.781,A -85,B 0,C 180,E1 -7272.958,E2 -7272.958} C_VEL
LIN {X 0,Y 477.362,Z 548.891,A -85,B 0,C 180,E1 -7273.661,E2 -7273.661} C_VEL
LIN {X 0,Y 476.739,Z 561.254,A -85,B 0,C 180,E1 -7274.502,E2 -7274.502} C_VEL
LIN {X 0,Y 476.094,Z 572.766,A -85,B 0,C 180,E1 -7275.466,E2 -7275.466} C_VEL
LIN {X 0,Y 475.543,Z 583.342,A -85,B 0,C 180,E1 -7276.539,E2 -7276.539} C_VEL
LIN {X 0,Y 475.062,Z 593.969,A -85,B 0,C 180,E1 -7277.844,E2 -7277.844} C_VEL
LIN {X 0,Y 474.588,Z 602.532,A -85,B 0,C 180,E1 -7279.116,E2 -7279.116} C_VEL
LIN {X 0,Y 474.234,Z 610.848,A -85,B 0,C 180,E1 -7280.617,E2 -7280.617} C_VEL
LIN {X 0,Y 473.994,Z 616.656,A -85,B 0,C 180,E1 -7281.902,E2 -7281.902} C_VEL
LIN {X 0,Y 473.888,Z 621.425,A -85,B 0,C 180,E1 -7283.185,E2 -7283.185} C_VEL
LIN {X 0,Y 473.821,Z 626.362,A -85,B 0,C 180,E1 -7284.893,E2 -7284.893} C_VEL
LIN {X 0,Y 473.787,Z 629.793,A -85,B 0,C 180,E1 -7286.598,E2 -7286.598} C_VEL
LIN {X 0,Y 473.722,Z 631.819,A -85,B 0,C 180,E1 -7288.299,E2 -7288.299} C_VEL
LIN {X 0,Y 473.668,Z 632.487,A -85,B 0,C 180,E1 -7289.999,E2 -7289.999} C_VEL
LIN {X 0,Y 473.721,Z 631.811,A -85,B 0,C 180,E1 -7291.7,E2 -7291.7} C_VEL
LIN {X 0,Y 473.786,Z 629.778,A -85,B 0,C 180,E1 -7293.401,E2 -7293.401} C_VEL
LIN {X 0,Y 473.821,Z 626.338,A -85,B 0,C 180,E1 -7295.105,E2 -7295.105} C_VEL
LIN {X 0,Y 473.89,Z 621.392,A -85,B 0,C 180,E1 -7296.813,E2 -7296.813} C_VEL
LIN {X 0,Y 474.075,Z 614.798,A -85,B 0,C 180,E1 -7298.524,E2 -7298.524} C_VEL
LIN {X 0,Y 474.328,Z 607.465,A -85,B 0,C 180,E1 -7300.025,E2 -7300.025} C_VEL
LIN {X 0,Y 474.808,Z 598.393,A -85,B 0,C 180,E1 -7301.526,E2 -7301.526} C_VEL
LIN {X 0,Y 475.269,Z 588.877,A -85,B 0,C 180,E1 -7302.815,E2 -7302.815} C_VEL
LIN {X 0,Y 475.77,Z 578.349,A -85,B 0,C 180,E1 -7303.997,E2 -7303.997} C_VEL
LIN {X 0,Y 476.477,Z 566.77,A -85,B 0,C 180,E1 -7305.067,E2 -7305.067} C_VEL
LIN {X 0,Y 477.157,Z 553.939,A -85,B 0,C 180,E1 -7306.031,E2 -7306.031} C_VEL
LIN {X 0,Y 477.785,Z 541.03,A -85,B 0,C 180,E1 -7306.8,E2 -7306.8} C_VEL
LIN {X 0,Y 478.291,Z 527.141,A -85,B 0,C 180,E1 -7307.437,E2 -7307.437} C_VEL
LIN {X 0,Y 478.807,Z 513.139,A -85,B 0,C 180,E1 -7307.892,E2 -7307.892} C_VEL
LIN {X 0,Y 479.12,Z 498.432,A -85,B 0,C 180,E1 -7308.189,E2 -7308.189} C_VEL
LIN {X 0,Y 480.096,Z 389.32,A -85,B 0,C 180,E1 -7309.858,E2 -7309.858} C_VEL
LIN {X 0,Y 476.452,Z 368.324,A -85,B 0,C 180,E1 -7310.361,E2 -7310.361} C_VEL
LIN {X 0,Y 477.247,Z 351.487,A -85,B 0,C 180,E1 -7312.969,E2 -7312.969} C_VEL
LIN {X 0,Y 478.007,Z 335.733,A -85,B 0,C 180,E1 -7315.45,E2 -7315.45} C_VEL
LIN {X 0,Y 475.569,Z 323.864,A -85,B 0,C 180,E1 -7317.54,E2 -7317.54} C_VEL
LIN {X 0,Y 474.675,Z 319.985,A -85,B 0,C 180,E1 -7318.279,E2 -7318.279} C_VEL
LIN {X 0,Y 474.597,Z 319.994,A -85,B 0,C 180,E1 -7321.217,E2 -7321.217} C_VEL
LIN {X 0,Y 474.631,Z 319.984,A -85,B 0,C 180,E1 -7324.24,E2 -7324.24} C_VEL
LIN {X 0,Y 474.589,Z 319.993,A -85,B 0,C 180,E1 -7327.383,E2 -7327.383} C_VEL
LIN {X 0,Y 474.644,Z 319.984,A -85,B 0,C 180,E1 -7329.65,E2 -7329.65} C_VEL
LIN {X 0,Y 474.611,Z 319.992,A -85,B 0,C 180,E1 -7332.933,E2 -7332.933} C_VEL
LIN {X 0,Y 474.61,Z 319.982,A -85,B 0,C 180,E1 -7335.895,E2 -7335.895} C_VEL
LIN {X 0,Y 474.627,Z 319.984,A -85,B 0,C 180,E1 -7339.039,E2 -7339.039} C_VEL
LIN {X 0,Y 474.605,Z 319.985,A -85,B 0,C 180,E1 -7341.703,E2 -7341.703} C_VEL
LIN {X 0,Y 474.623,Z 319.99,A -85,B 0,C 180,E1 -7344.725,E2 -7344.725} C_VEL
LIN {X 0,Y 474.63,Z 319.983,A -85,B 0,C 180,E1 -7347.787,E2 -7347.787} C_VEL
LIN {X 0,Y 474.626,Z 319.986,A -85,B 0,C 180,E1 -7350.882,E2 -7350.882} C_VEL
LIN {X 0,Y 474.657,Z 319.98,A -85,B 0,C 180,E1 -7353.628,E2 -7353.628} C_VEL
LIN {X 0,Y 474.628,Z 319.983,A -85,B 0,C 180,E1 -7356.641,E2 -7356.641} C_VEL
LIN {X 0,Y 474.647,Z 319.987,A -85,B 0,C 180,E1 -7360.089,E2 -7360.089} C_VEL
LIN {X 0,Y 474.642,Z 319.984,A -85,B 0,C 180,E1 -7362.774,E2 -7362.774} C_VEL
LIN {X 0,Y 474.639,Z 319.98,A -85,B 0,C 180,E1 -7365.42,E2 -7365.42} C_VEL
LIN {X 0,Y 474.695,Z 319.979,A -85,B 0,C 180,E1 -7368.037,E2 -7368.037} C_VEL
LIN {X 0,Y 474.717,Z 319.977,A -85,B 0,C 180,E1 -7371.486,E2 -7371.486} C_VEL
LIN {X 0,Y 474.758,Z 319.974,A -85,B 0,C 180,E1 -7374.052,E2 -7374.052} C_VEL
LIN {X 0,Y 474.87,Z 319.955,A -85,B 0,C 180,E1 -7377.455,E2 -7377.455} C_VEL
LIN {X 0,Y 474.869,Z 319.957,A -85,B 0,C 180,E1 -7380,E2 -7380} C_VEL
LIN {X 0,Y 474.871,Z 319.954,A -85,B 0,C 180,E1 -7382.544,E2 -7382.544} C_VEL
LIN {X 0,Y 474.718,Z 319.977,A -85,B 0,C 180,E1 -7385.948,E2 -7385.948} C_VEL
LIN {X 0,Y 474.656,Z 319.979,A -85,B 0,C 180,E1 -7388.515,E2 -7388.515} C_VEL
LIN {X 0,Y 474.693,Z 319.976,A -85,B 0,C 180,E1 -7391.962,E2 -7391.962} C_VEL
LIN {X 0,Y 474.668,Z 319.98,A -85,B 0,C 180,E1 -7395.767,E2 -7395.767} C_VEL
LIN {X 0,Y 474.648,Z 319.986,A -85,B 0,C 180,E1 -7399.011,E2 -7399.011} C_VEL
LIN {X 0,Y 474.577,Z 319.991,A -85,B 0,C 180,E1 -7401.729,E2 -7401.729} C_VEL
LIN {X 0,Y 474.616,Z 319.987,A -85,B 0,C 180,E1 -7404.495,E2 -7404.495} C_VEL
LIN {X 0,Y 474.627,Z 319.986,A -85,B 0,C 180,E1 -7407.324,E2 -7407.324} C_VEL
LIN {X 0,Y 474.587,Z 319.992,A -85,B 0,C 180,E1 -7410.231,E2 -7410.231} C_VEL
LIN {X 0,Y 474.615,Z 319.989,A -85,B 0,C 180,E1 -7413.222,E2 -7413.222} C_VEL
LIN {X 0,Y 474.579,Z 319.993,A -85,B 0,C 180,E1 -7416.324,E2 -7416.324} C_VEL
LIN {X 0,Y 474.608,Z 319.987,A -85,B 0,C 180,E1 -7419.647,E2 -7419.647} C_VEL
LIN {X 0,Y 474.615,Z 319.986,A -85,B 0,C 180,E1 -7422.237,E2 -7422.237} C_VEL
LIN {X 0,Y 474.608,Z 319.99,A -85,B 0,C 180,E1 -7425.298,E2 -7425.298} C_VEL
LIN {X 0,Y 474.631,Z 320.01,A -85,B 0,C 180,E1 -7428.436,E2 -7428.436} C_VEL
LIN {X 0,Y 476.764,Z 330.689,A -85,B 0,C 180,E1 -7430.666,E2 -7430.666} C_VEL
LIN {X 0,Y 476.679,Z 336.102,A -85,B 0,C 180,E1 -7431.712,E2 -7431.712} C_VEL
LIN {X 0,Y 480.361,Z 352.774,A -85,B 0,C 180,E1 -7432.152,E2 -7432.152} C_VEL
LIN {X 0,Y 479.192,Z 471.943,A -85,B 0,C 180,E1 -7433.995,E2 -7433.995} C_VEL
LIN {X 0,Y 479.009,Z 480.995,A -85,B 0,C 180,E1 -7434.221,E2 -7434.221} C_VEL
LIN {X 0,Y 477.824,Z 488.577,A -85,B 0,C 180,E1 -7434.423,E2 -7434.423} C_VEL
LIN {X 0,Y 475.187,Z 495.931,A -85,B 0,C 180,E1 -7434.61,E2 -7434.61} C_VEL
LIN {X 0,Y 472.063,Z 505.046,A -85,B 0,C 180,E1 -7434.92,E2 -7434.92} C_VEL
LIN {X 0,Y 471.228,Z 510.399,A -85,B 0,C 180,E1 -7435.189,E2 -7435.189} C_VEL
LIN {X 0,Y 470.669,Z 522.179,A -85,B 0,C 180,E1 -7435.949,E2 -7435.949} C_VEL
LIN {X 0,Y 469.956,Z 533.814,A -85,B 0,C 180,E1 -7436.872,E2 -7436.872} C_VEL
LIN {X 0,Y 469.299,Z 545.489,A -85,B 0,C 180,E1 -7438.012,E2 -7438.012} C_VEL
LIN {X 0,Y 468.711,Z 555.084,A -85,B 0,C 180,E1 -7439.145,E2 -7439.145} C_VEL
LIN {X 0,Y 468.1,Z 564.899,A -85,B 0,C 180,E1 -7440.551,E2 -7440.551} C_VEL
LIN {X 0,Y 467.611,Z 573.117,A -85,B 0,C 180,E1 -7441.988,E2 -7441.988} C_VEL
LIN {X 0,Y 467.301,Z 578.823,A -85,B 0,C 180,E1 -7443.181,E2 -7443.181} C_VEL
LIN {X 0,Y 467.033,Z 584.164,A -85,B 0,C 180,E1 -7444.54,E2 -7444.54} C_VEL
LIN {X 0,Y 466.869,Z 588.816,A -85,B 0,C 180,E1 -7446.019,E2 -7446.019} C_VEL
LIN {X 0,Y 466.761,Z 591.194,A -85,B 0,C 180,E1 -7446.954,E2 -7446.954} C_VEL
LIN {X 0,Y 466.659,Z 593.137,A -85,B 0,C 180,E1 -7447.884,E2 -7447.884} C_VEL
LIN {X 0,Y 466.614,Z 594.934,A -85,B 0,C 180,E1 -7449.038,E2 -7449.038} C_VEL
LIN {X 0,Y 466.57,Z 596.484,A -85,B 0,C 180,E1 -7450.648,E2 -7450.648} C_VEL
LIN {X 0,Y 466.565,Z 596.852,A -85,B 0,C 180,E1 -7452.467,E2 -7452.467} C_VEL
LIN {X 0,Y 466.574,Z 595.791,A -85,B 0,C 180,E1 -7454.269,E2 -7454.269} C_VEL
LIN {X 0,Y 466.647,Z 593.315,A -85,B 0,C 180,E1 -7456.057,E2 -7456.057} C_VEL
LIN {X 0,Y 466.856,Z 589.367,A -85,B 0,C 180,E1 -7457.834,E2 -7457.834} C_VEL
LIN {X 0,Y 467.04,Z 583.828,A -85,B 0,C 180,E1 -7459.598,E2 -7459.598} C_VEL
LIN {X 0,Y 467.374,Z 577.565,A -85,B 0,C 180,E1 -7461.134,E2 -7461.134} C_VEL
LIN {X 0,Y 467.746,Z 570.181,A -85,B 0,C 180,E1 -7462.595,E2 -7462.595} C_VEL
LIN {X 0,Y 468.271,Z 561.682,A -85,B 0,C 180,E1 -7463.97,E2 -7463.97} C_VEL
LIN {X 0,Y 468.802,Z 551.958,A -85,B 0,C 180,E1 -7465.271,E2 -7465.271} C_VEL
LIN {X 0,Y 469.375,Z 541.199,A -85,B 0,C 180,E1 -7466.46,E2 -7466.46} C_VEL
LIN {X 0,Y 470.098,Z 529.248,A -85,B 0,C 180,E1 -7467.537,E2 -7467.537} C_VEL
LIN {X 0,Y 470.705,Z 517.599,A -85,B 0,C 180,E1 -7468.39,E2 -7468.39} C_VEL
LIN {X 0,Y 471.345,Z 504.633,A -85,B 0,C 180,E1 -7469.146,E2 -7469.146} C_VEL
LIN {X 0,Y 471.822,Z 490.732,A -85,B 0,C 180,E1 -7469.761,E2 -7469.761} C_VEL
LIN {X 0,Y 472.209,Z 477.051,A -85,B 0,C 180,E1 -7470.187,E2 -7470.187} C_VEL
LIN {X 0,Y 472.447,Z 460.171,A -85,B 0,C 180,E1 -7470.507,E2 -7470.507} C_VEL
LIN {X 0,Y 473.364,Z 352.607,A -85,B 0,C 180,E1 -7472.172,E2 -7472.172} C_VEL
LIN {X 0,Y 469.696,Z 336.046,A -85,B 0,C 180,E1 -7472.6,E2 -7472.6} C_VEL
LIN {X 0,Y 469.776,Z 331.711,A -85,B 0,C 180,E1 -7473.431,E2 -7473.431} C_VEL
LIN {X 0,Y 467.735,Z 320.85,A -85,B 0,C 180,E1 -7475.66,E2 -7475.66} C_VEL
LIN {X 0,Y 467.665,Z 320.857,A -85,B 0,C 180,E1 -7478.644,E2 -7478.644} C_VEL
LIN {X 0,Y 467.654,Z 320.852,A -85,B 0,C 180,E1 -7482.146,E2 -7482.146} C_VEL
LIN {X 0,Y 467.647,Z 320.854,A -85,B 0,C 180,E1 -7485.885,E2 -7485.885} C_VEL
LIN {X 0,Y 467.62,Z 320.863,A -85,B 0,C 180,E1 -7489.309,E2 -7489.309} C_VEL
LIN {X 0,Y 467.529,Z 320.868,A -85,B 0,C 180,E1 -7492.075,E2 -7492.075} C_VEL
LIN {X 0,Y 467.554,Z 320.87,A -85,B 0,C 180,E1 -7494.891,E2 -7494.891} C_VEL
LIN {X 0,Y 467.542,Z 320.867,A -85,B 0,C 180,E1 -7497.775,E2 -7497.775} C_VEL
LIN {X 0,Y 467.534,Z 320.875,A -85,B 0,C 180,E1 -7501.039,E2 -7501.039} C_VEL
LIN {X 0,Y 467.563,Z 320.864,A -85,B 0,C 180,E1 -7504.238,E2 -7504.238} C_VEL
LIN {X 0,Y 467.513,Z 320.874,A -85,B 0,C 180,E1 -7507.181,E2 -7507.181} C_VEL
LIN {X 0,Y 467.554,Z 320.866,A -85,B 0,C 180,E1 -7510.268,E2 -7510.268} C_VEL
LIN {X 0,Y 467.516,Z 320.875,A -85,B 0,C 180,E1 -7512.569,E2 -7512.569} C_VEL
LIN {X 0,Y 467.561,Z 320.868,A -85,B 0,C 180,E1 -7515.052,E2 -7515.052} C_VEL
LIN {X 0,Y 467.554,Z 320.873,A -85,B 0,C 180,E1 -7518.727,E2 -7518.727} C_VEL
LIN {X 0,Y 467.536,Z 320.868,A -85,B 0,C 180,E1 -7521.953,E2 -7521.953} C_VEL
